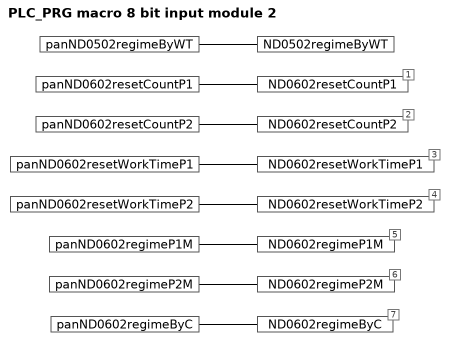
[picture p72: PLC_PRG macro 8 bit input module 2 (CFC)]
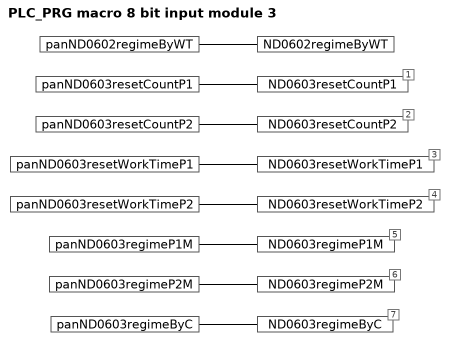
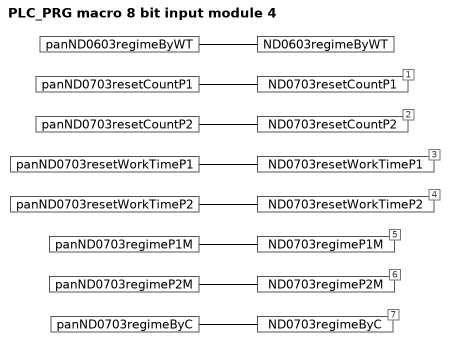
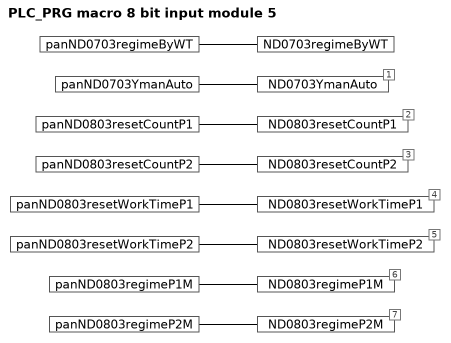
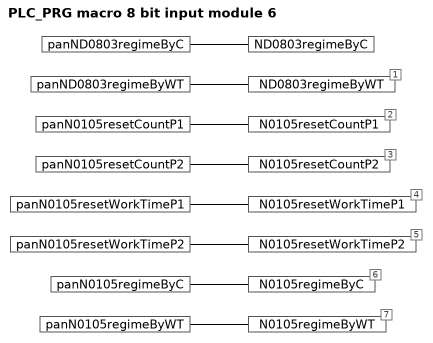
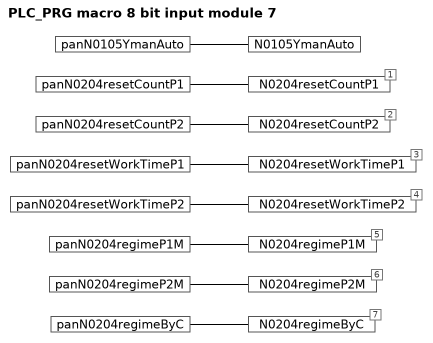
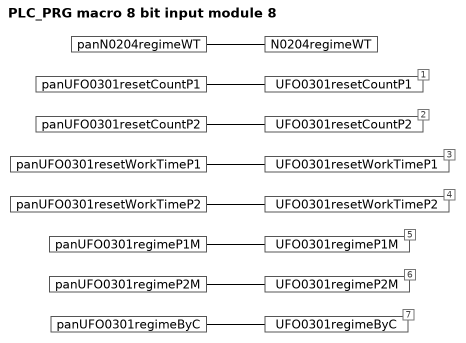
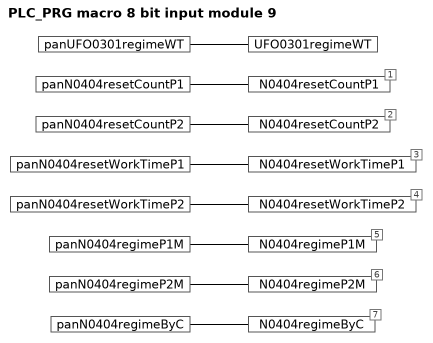
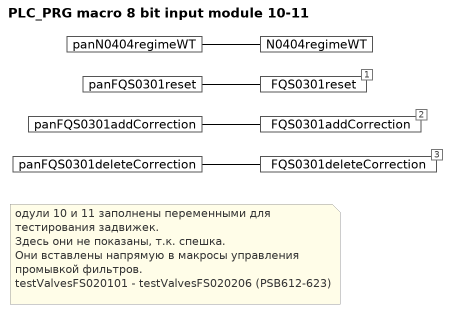
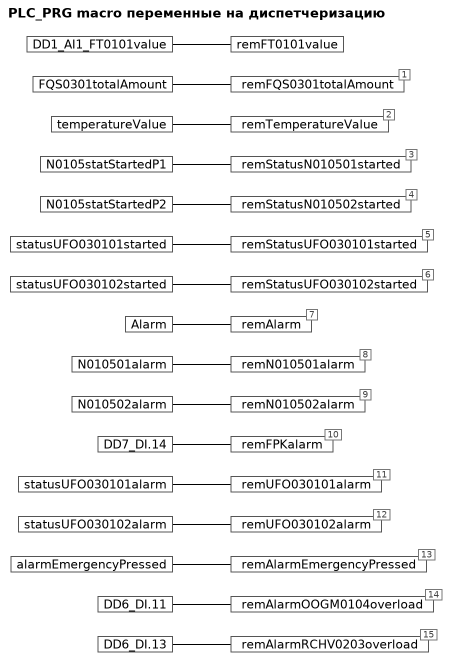
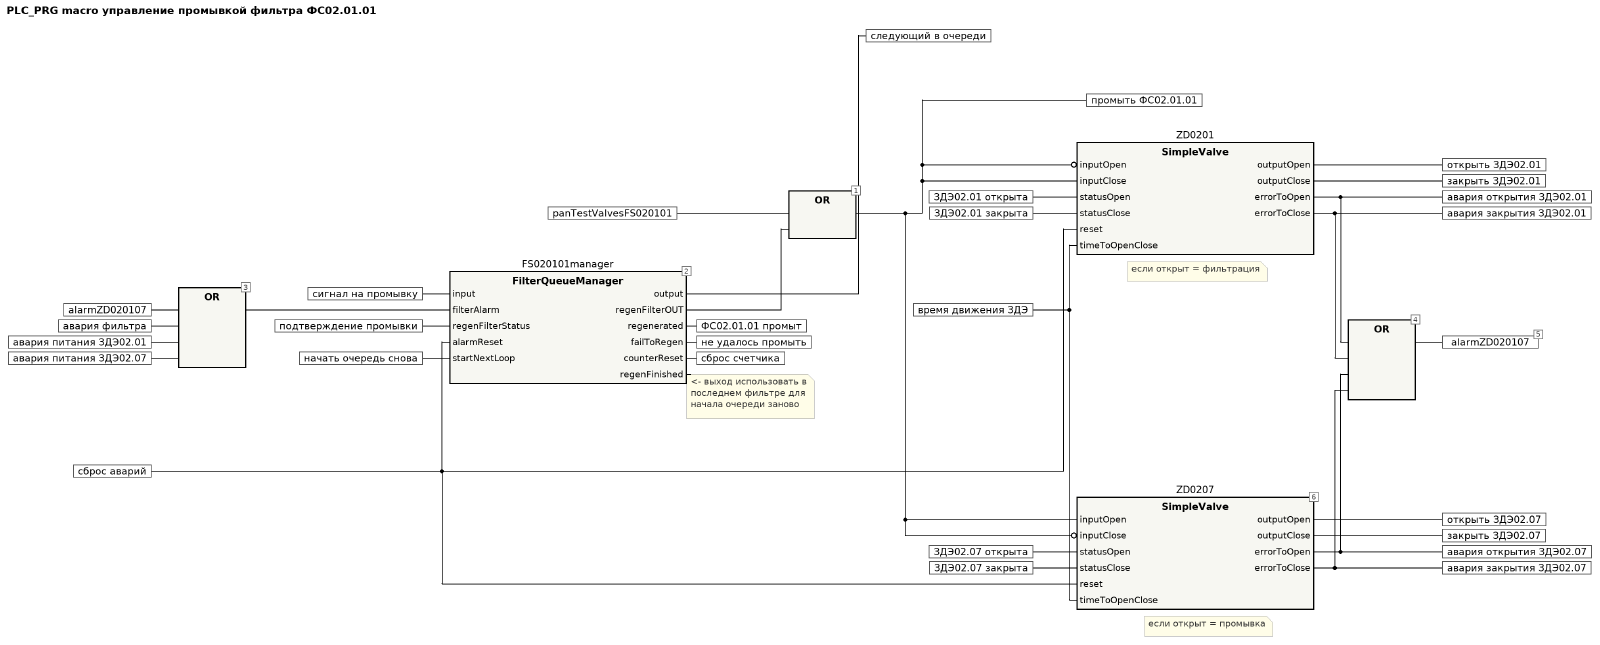
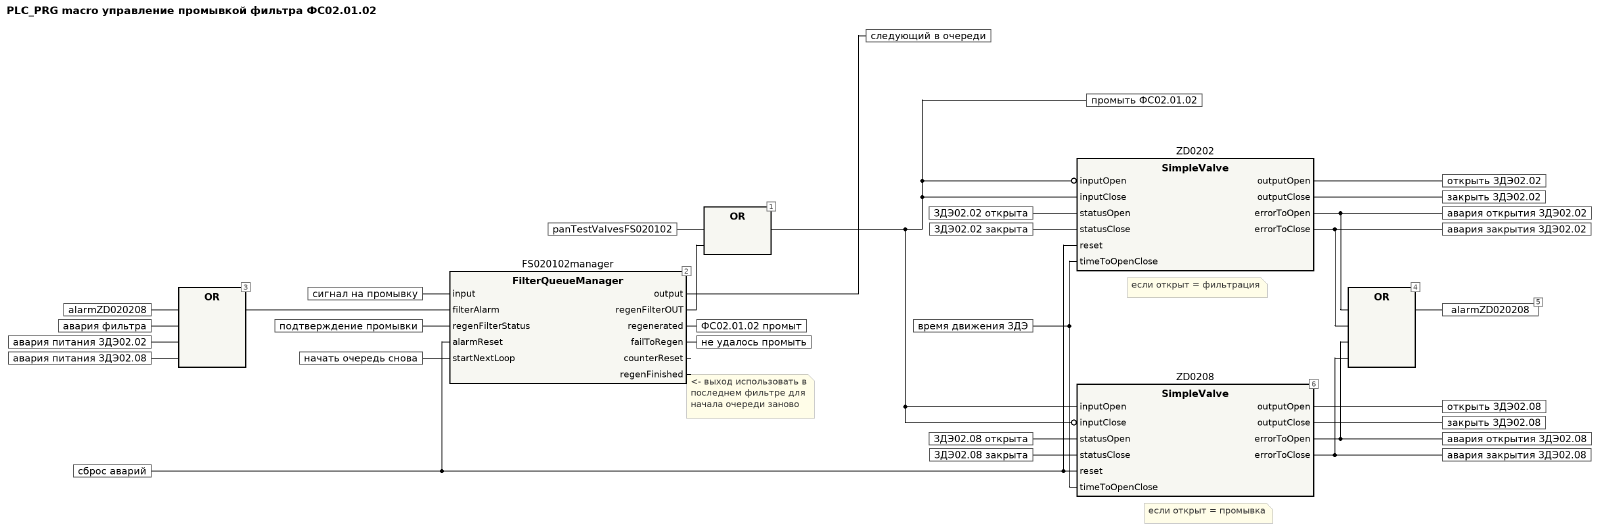
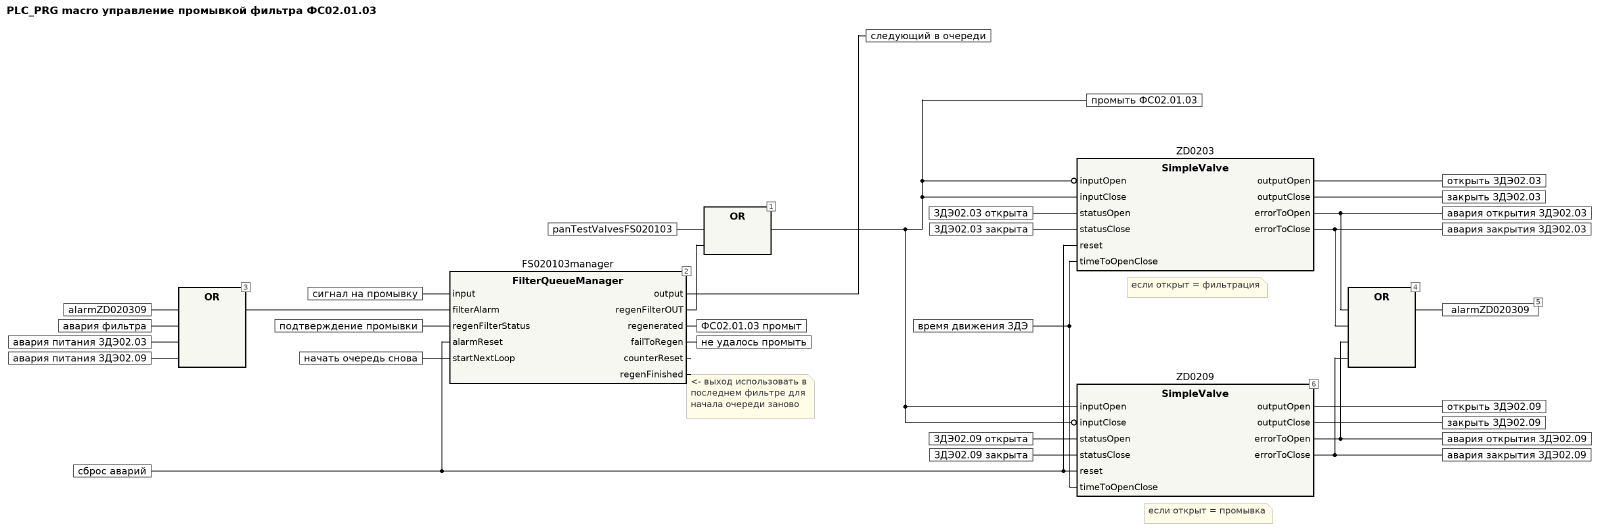
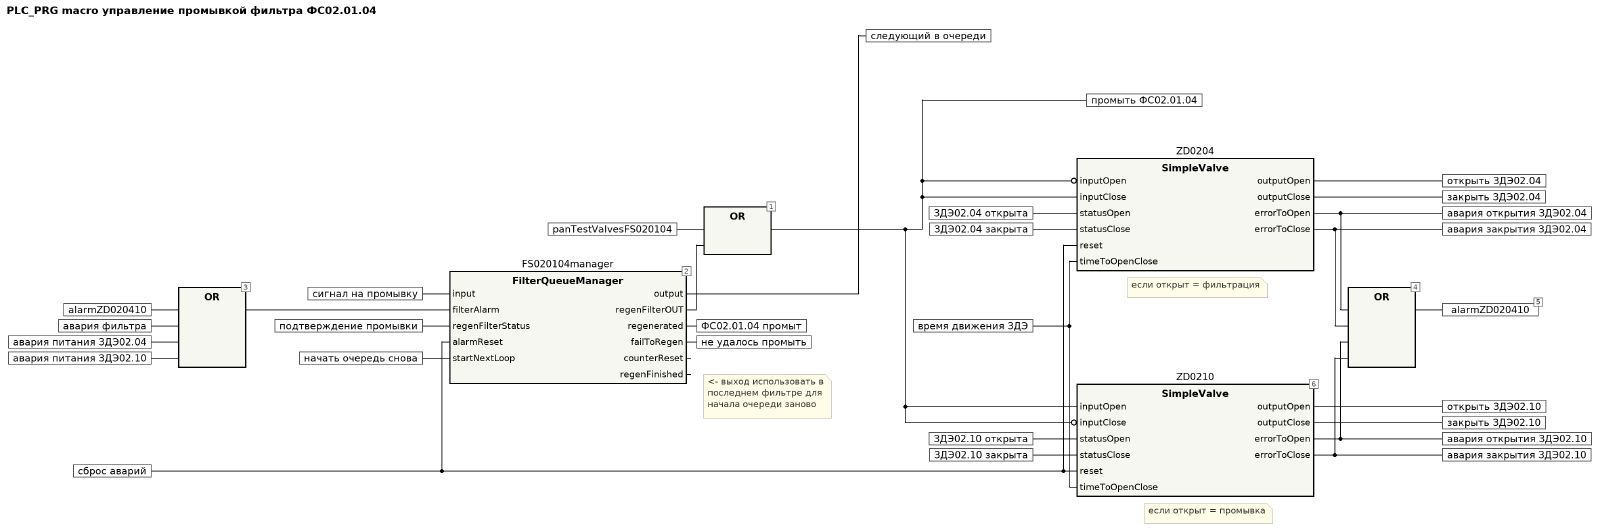
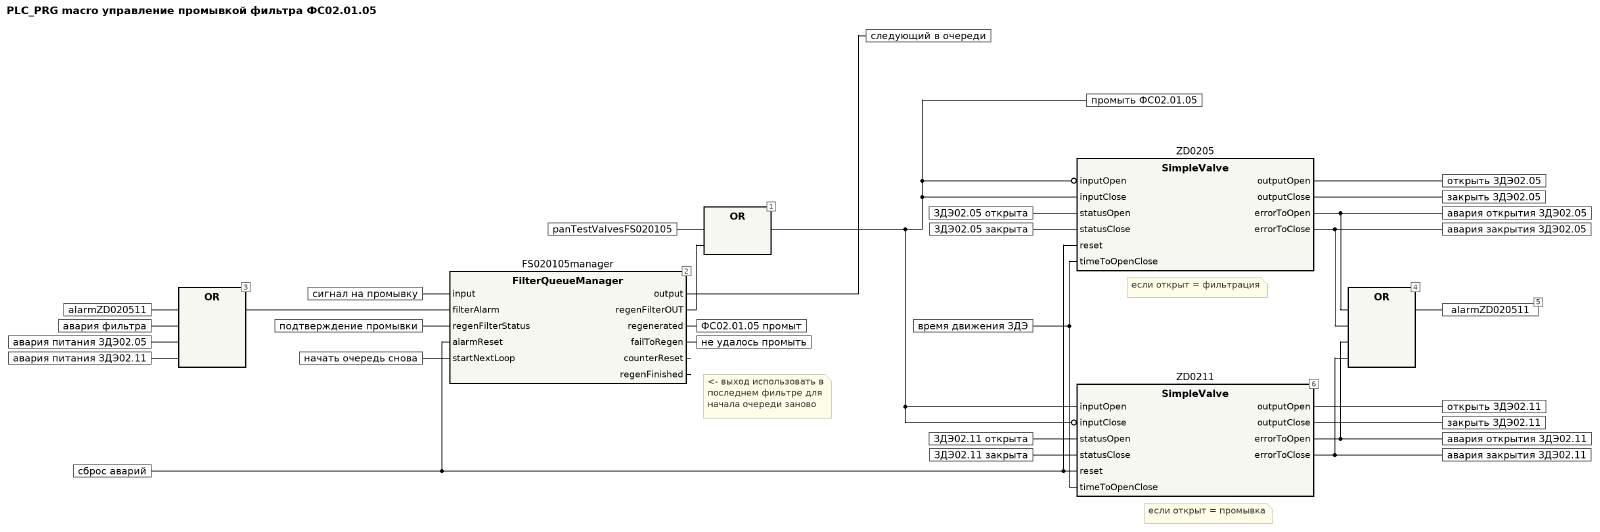
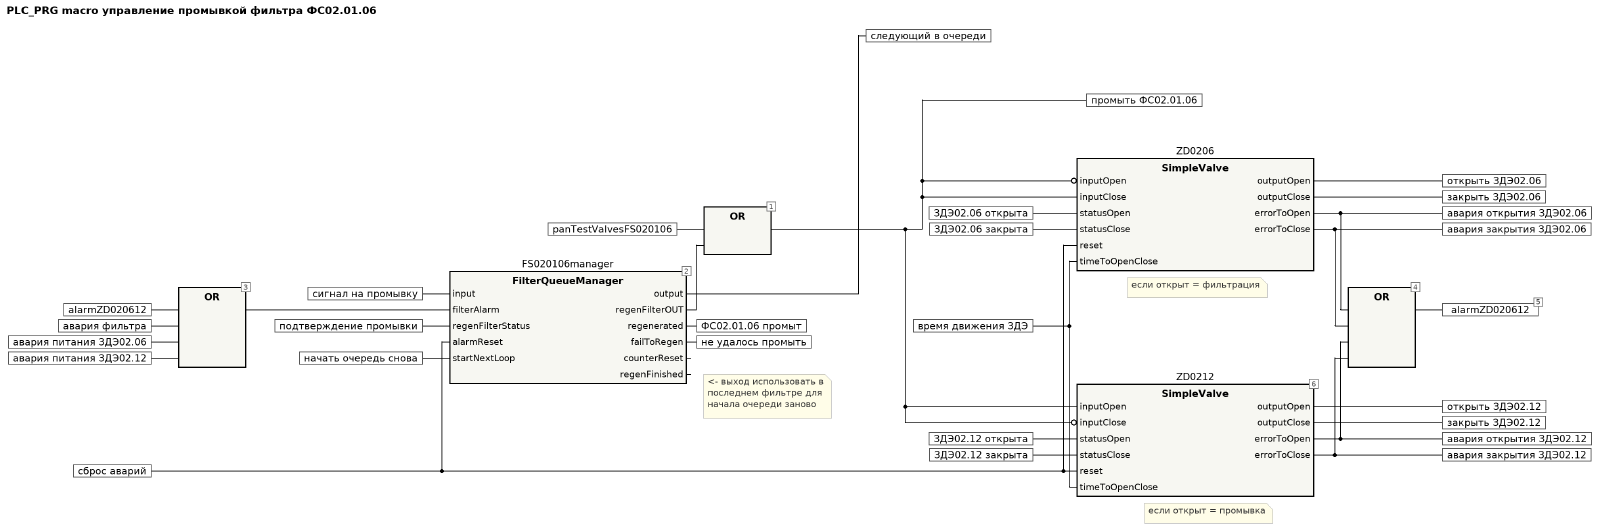
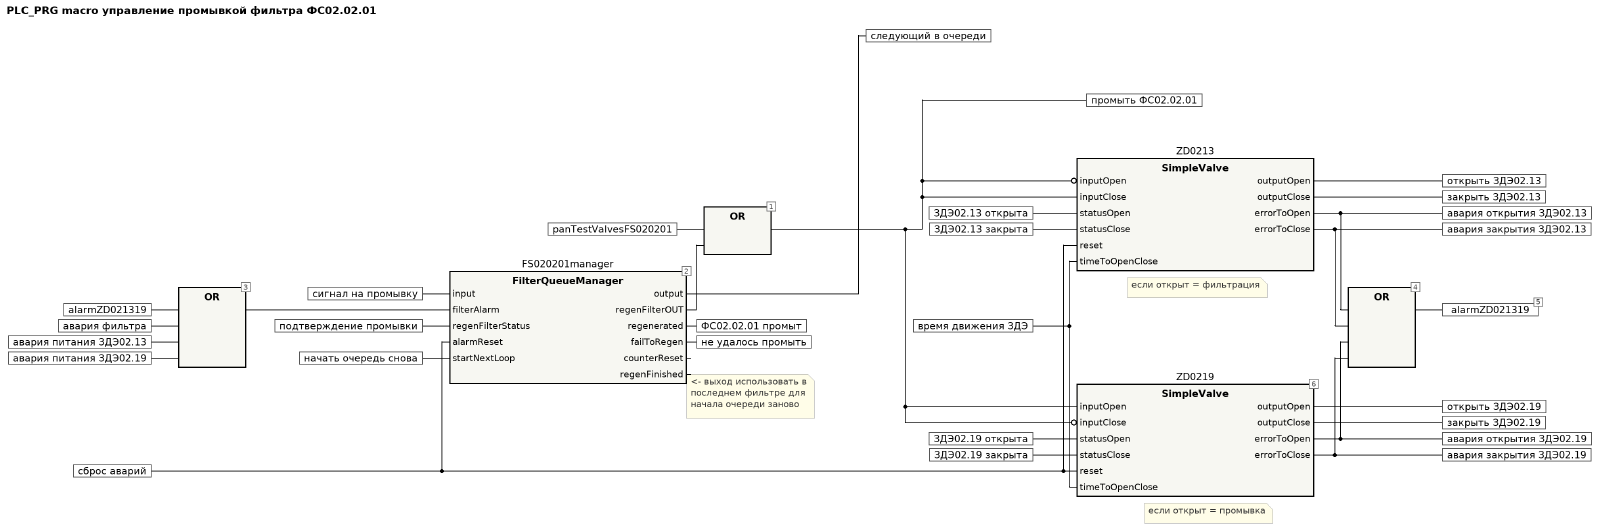
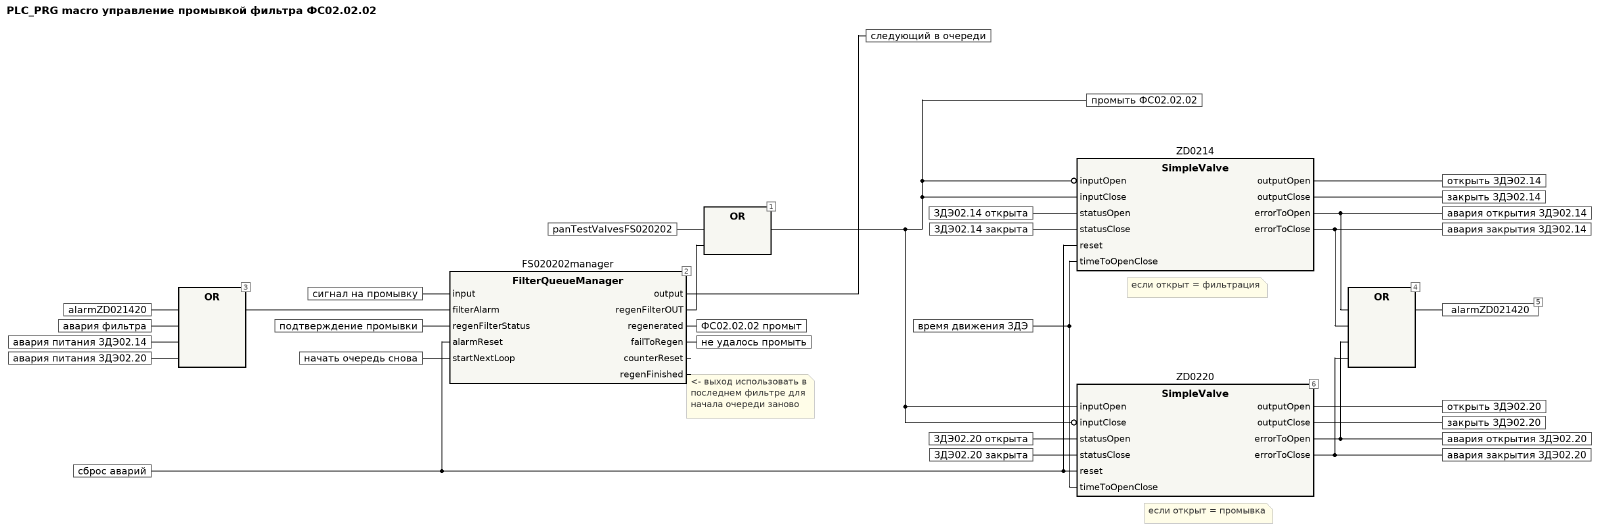
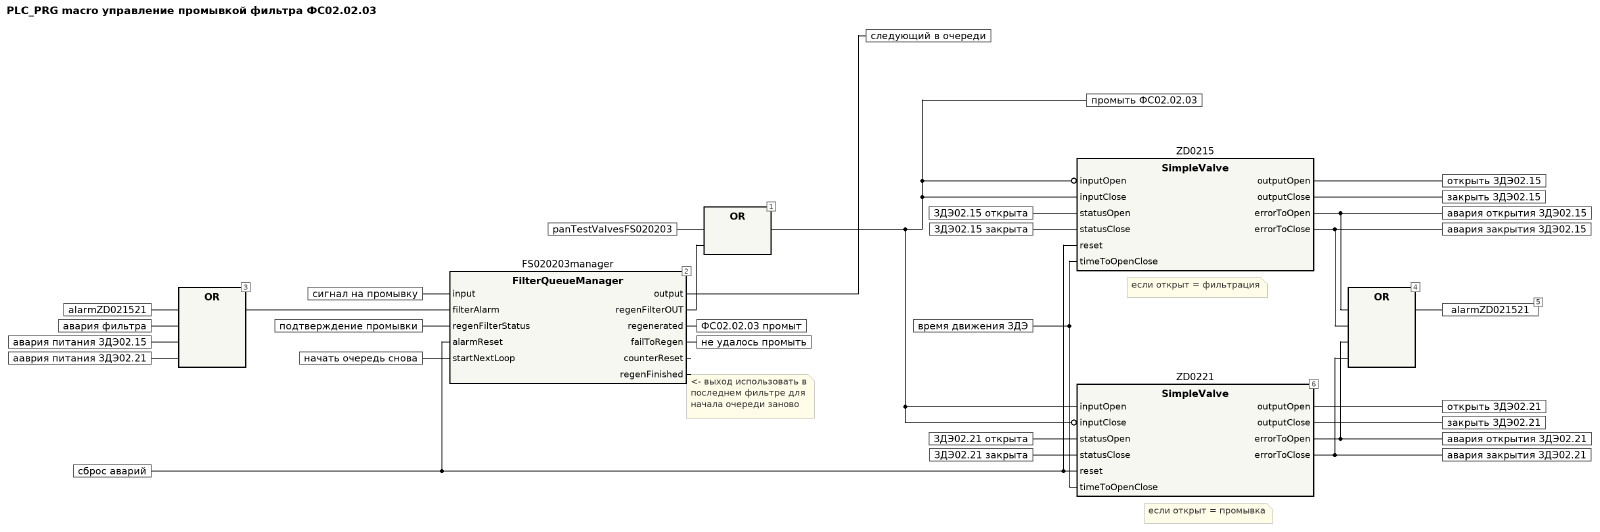
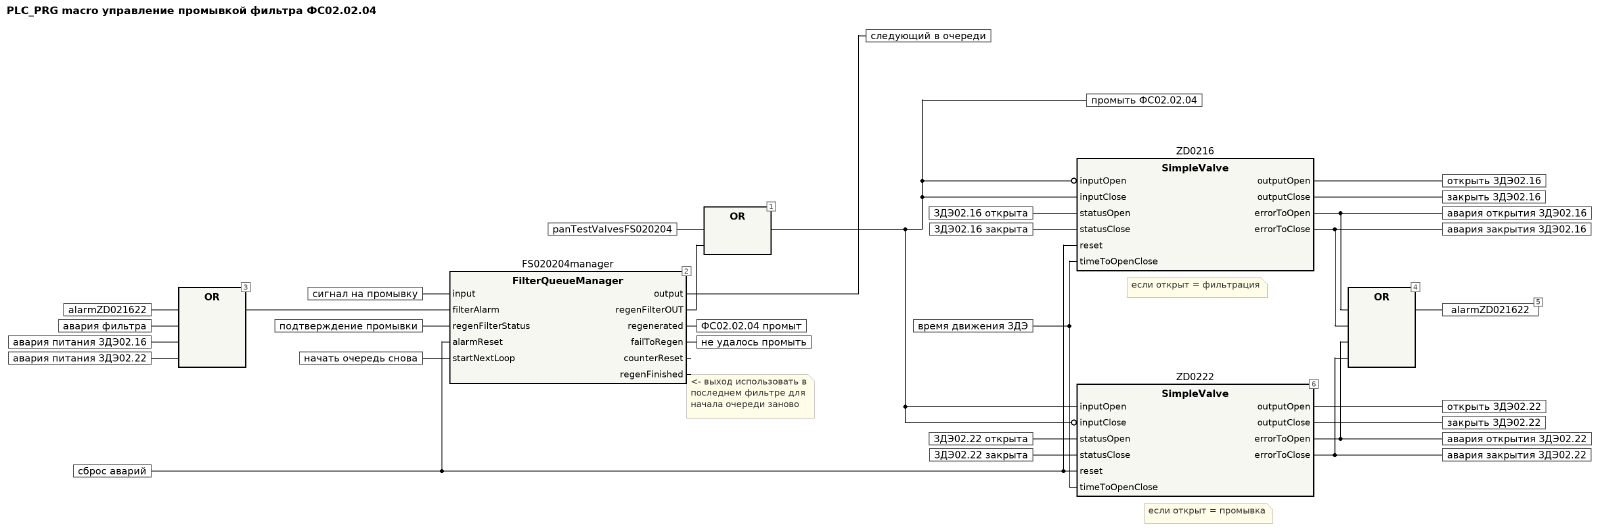
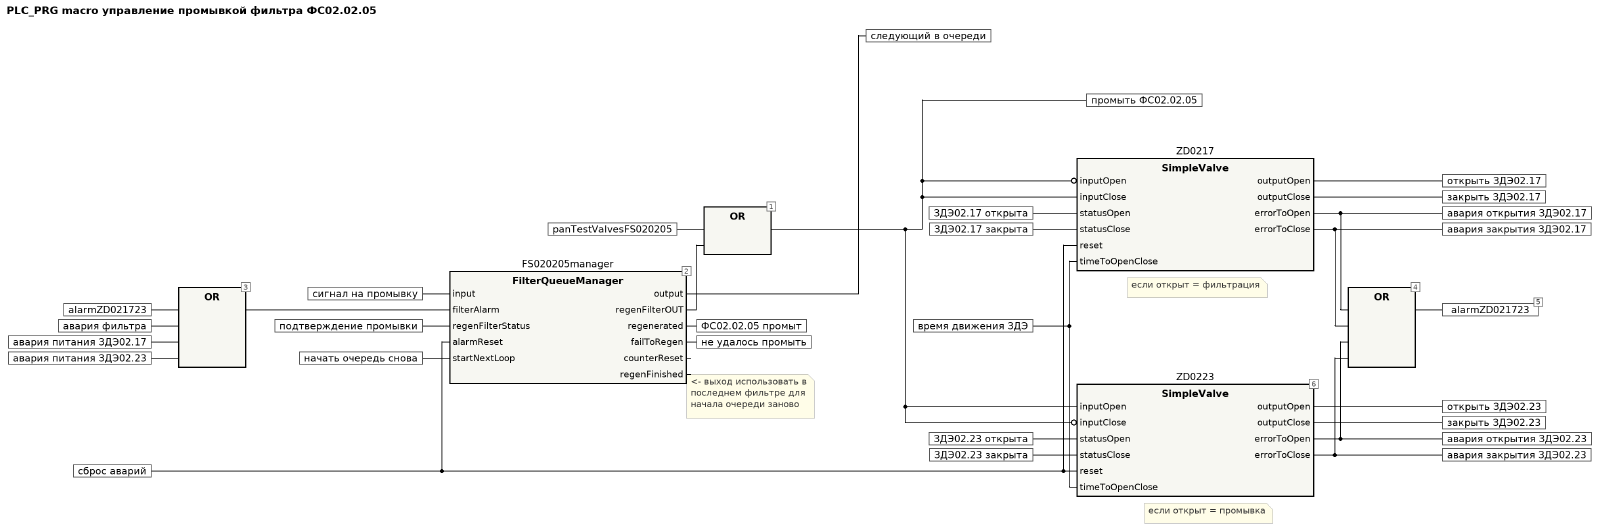
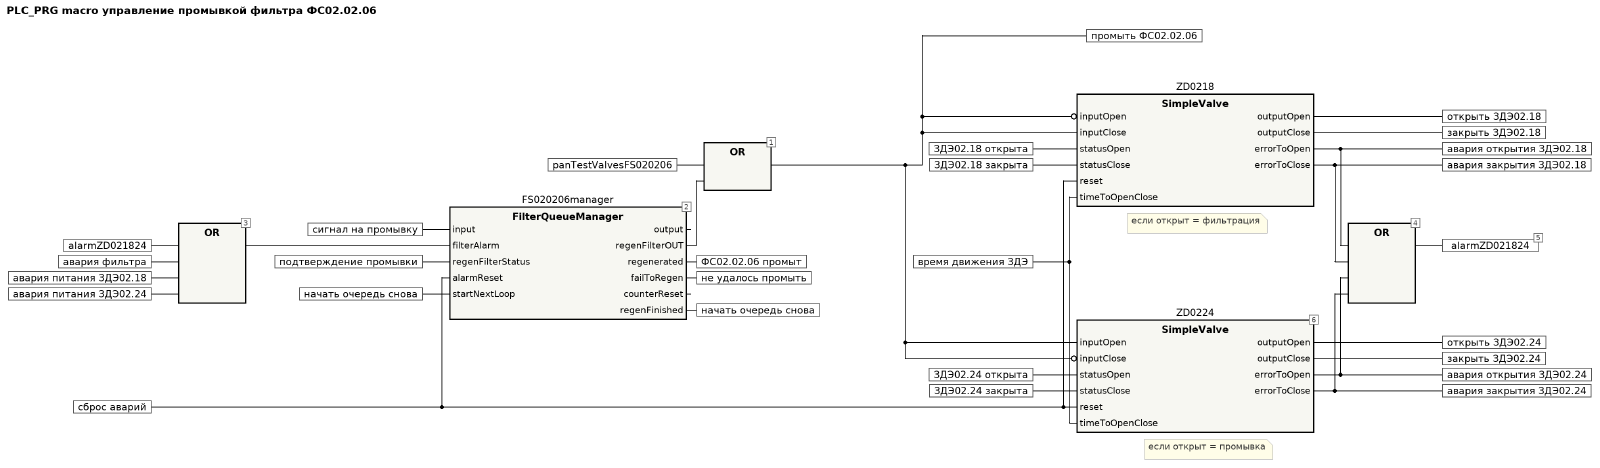
_CFC_ (* Continuous Function Chart, elements in execution order *)
(* 0 = перелив *)
(* авария обоих УФО, если проблемы / открытия/закрытия на одной из задвижек *)
(* авария питания ЗДЭ03.02 *)
(* авария питания ЗДЭ03.01 *)
(* статус-пуск Н01.05/02 *)
(* вкл КМ3 *)
(* Статус ПУСК / ЧРП Н01.05 *)
(* статус-пуск Н01.05/01 *)
(* вкл КМ2 *)
(* контроль обрыва или ошибок модулей в сети ПЛК *)
(* LSA01.02 перелив ОГМ01.04 *)
(* Нажат аварийный стоп. *)
(* авария сети (РКФ) *)
(* разрешение работы КНС / 1 = разрешено *)
(* Нажат аварийный стоп. *)
(* Блок управления разрешением работы КНС *)
(* авария сети (РКФ) *)
(* Авария питания клапанов КЭМ. *)
(* Авария питания розеток / управл.клапанов фильтров. *)
(* авария КНС *)
(* блок подачи сигнала на промывку *)
(* суммируем каждую секунду значение / мгновенного расхода в кубометрах в секунду *)
(* преобразуем расход из / кубометров в час в / кубометры в секунду *)
(* если есть расход / (больше нуля) *)
(* выдает импульс / каждую секунду *)
(* здесь мгновенный расход / в кубометрах в час (FT01.02) *)
(* Авария Н02.04/01 (0=авария) *)
(* Авария Н02.04/02 (0=авария) *)
(* промывка ФС02.01/06 *)
(* промывка ФС02.01/05 *)
(* промывка ФС02.01/04 *)
(* промывка ФС02.01/03 *)
(* промывка ФС02.01/02 *)
(* промывка ФС02.01/01 *)
(* пуск/стоп НД08.03/01 *)
(* пуск/стоп НД08.03/02 *)
(* пуск/стоп НД06.03/01 *)
(* пуск/стоп НД06.03/02 *)
(* пуск/стоп НД06.02/01 *)
(* пуск/стоп НД06.02/02 *)
(* пуск/стоп НД08.04 *)
(* пуск/стоп НД07.03/01 *)
(* пуск/стоп НД07.03/02 *)
(* авария М08.02 (УПФ) *)
(* авария М07.02 (УПЩ) *)
(* авария М06.04 (УПК) *)
(* работа М08.02 (УПФ) *)
(* работа М07.02 (УПЩ) *)
(* работа М06.04 (УПК) *)
(* Контроль, если УФО включили вручную, / а потока при этом нет. *)
(* авария УФО03.01/02 *)
(* работа УФО03.01/02 *)
(* авария УФО03.01/01 *)
(* Для подачи предостережения на пульте / оператора (при необходимости), а также / сигнализации лампой АВАРИЯ. *)
(* работа УФО03.01/01 *)
(* авария УФО03.01/02 *)
(* авария УФО03.01/01 *)
(* авария Н04.04/01 *)
(* авария Н04.04/02 *)
(* время контроля старта ФПК (по умолч.=3мин) *)
(* время работы ФПК после спада сигнала датч.осадка *)
(* запуск фильтрации *)
(* Защита от сухого хода насоса ФПК *)
(* датчик уровня осадка *)
(* Давление на входе ФПК (0...16 бар) *)
(* авария ФПК *)
(* подающий насос ФПК работает *)
(* ФПК готов к приему *)
(* ФПК не запустился *)
(* рН-метр QE01.02 на входе, / диапазон 0...14 *)
(* авария входа рН-метра QE01.01 *)
(* авария входа расходомера FT01.02 *)
(* расходомер FT01.01 на входе, / диапазон 0...600куб/час *)
(* авария НД08.04 *)
(* управление 4...20мА НД08.03/01 *)
(* пуск/стоп НД08.03/01 *)
(* пуск/стоп НД08.03/02 *)
(* управление 4...20мА НД08.03/02 *)
(* авария привода НД08.03/01 *)
(* авария привода НД08.03/02 *)
(* авария НД07.03/01 *)
(* авария НД07.03/02 *)
(* управление 4...20мА НД07.03/01 *)
(* управление 4...20мА НД07.03/02 *)
(* пуск/стоп НД07.03/01 *)
(* пуск/стоп НД07.03/02 *)
(* авария НД07.03/01 *)
(* авария НД07.03/02 *)
(* авария НД06.03/01 *)
(* авария НД06.03/02 *)
(* авария НД06.02/01 *)
(* авария НД06.02/02 *)
(* управление 4...20мА НД06.03/01 *)
(* пуск/стоп НД06.03/01 *)
(* пуск/стоп НД06.03/02 *)
(* управление 4...20мА НД06.03/02 *)
(* авария НД06.03/01 *)
(* авария НД06.03/02 *)
(* управление 4...20мА НД06.02/01 *)
(* пуск/стоп НД06.02/01 *)
(* пуск/стоп НД06.02/02 *)
(* управление 4...20мА НД06.02/02 *)
(* авария НД06.02/01 *)
(* авария НД06.02/02 *)
(* ошибка блока дозирования НД05.02 *)
(* авария входа датчика температуры *)
(* лампа АВАРИЯ *)
(* датчик температуры в помещении / (метран) диапазон: 0...+100С *)
(* управление 4...20мА НД05.02/01 *)
(* пуск/стоп НД05.02/01 *)
(* авария НД05.02/01 *)
(* авария НД05.02/02 *)
(* пуск/стоп НД05.02/02 *)
(* управление 4...20мА НД05.02/02 *)
(* АВАРИИ *)
(* авария привода НД08.03/01 *)
(* авария привода НД08.03/02 *)
(* авария НД08.04 *)
(* насос Н04.01 работает *)
(* пуск/стоп НД08.04 *)
(* управление 4...20мА НД08.04 *)
(* авария входа расходомера FT01.01 *)
(* расходомер FT01.02 на входе, / диапазон 0...600куб/час *)
(* рН-метр QE01.01 на входе, / диапазон 0...14 *)
(* авария входа рН-метра QE01.02 *)
(* сухой ход НД08.03/01 *)
(* сухой ход НД08.03/02 *)
(* сухой ход НД08.03/01 *)
(* сухой ход НД08.03/02 *)
(* LSA01.02 перелив ОГМ01.04 *)
(* Инициализирует требуемые булевые переменные / в момент старта выполнения программы. *)
(* Статус ПУСК ЧРП Н01.05 *)
(* LS01.03 - рабочий верхний уровень ОГМ01.04 автоматический пуск 01.05 *)
(* LS01.04 - нижний уровень ОГМ01.04, сухой ход Н01.05 *)
(* SA1 Ручной выбор Н01.05/01 = главный *)
(* SA1 Ручной выбор Н01.05/02 = главный *)
(* Стоп  Н01.05 (сброс самоподхвата реле) *)
(* время на создание потока *)
(* Пуск  Н01.05 *)
(* КМ1 питание ЧРП *)
(* КМ2 питание насоса 1 *)
(* КМ3 питание насоса 2 *)
(* Авария ЧРП Н01.05 *)
(* термоконтакт Н01.05/01 *)
(* термоконтакт Н01.05/02 *)
(* авария питания ЗДЭ02.25 *)
(* LSА02.01 Перелив РЧВ02.03 *)
(* Давление на входе ФПК / 0...16 бар (мах допуст.10) *)
(* Авария входа AI6 ПЛК, давл.ФПК *)
(* авария ФПК *)
(* Открыть КШЭ04.01 *)
(* статус КШЭ04.01 открыт *)
(* Закрыть КШЭ04.01 *)
(* статус КШЭ04.01 закрыт *)
(* подающий насос ФПК работает *)
(* стоп Н04.04 *)
(* пуск Н04.04/02 *)
(* пуск Н04.04/01 *)
(* авт.пуск Н04.04 *)
(* сухой ход Н04.04, 0=защита *)
(* авария Н04.04/01, 0=авария *)
(* авария Н04.04/02, 0=авария *)
(* импульсный расходомер *)
(* Авария Н02.04/01 (0=авария) *)
(* Авария Н02.04/02 (0=авария) *)
(* промывка ФС02.02/06 *)
(* промывка ФС02.02/05 *)
(* промывка ФС02.02/04 *)
(* промывка ФС02.02/03 *)
(* промывка ФС02.02/02 *)
(* промывка ФС02.02/01 *)
(* Клапан КЭМ05.01 открыт. *)
(* Клапан КЭМ06.01 открыт. *)
(* Клапан КЭМ07.01 открыт. *)
(* Клапан КЭМ08.01 открыт. *)
(* Сухой ход Н02.04 (LS02.03) 0=сух.ход *)
(* Стоп Н02.04 *)
(* Пуск Н02.04/01 *)
(* Пуск Н02.04/02 *)
(* текущий объем *)
(* заданный до промывки объем *)
(* 0=авария *)
(* авария (при 0) ФС02.01/06 *)
(* авария (при 0) ФС02.01/05 *)
(* авария (при 0) ФС02.01/04 *)
(* авария (при 0) ФС02.01/03 *)
(* авария (при 0) ФС02.01/02 *)
(* авария (при 0) ФС02.01/01 *)
(* авария (при 0) ФС02.02/06 *)
(* авария (при 0) ФС02.02/05 *)
(* авария (при 0) ФС02.02/04 *)
(* авария (при 0) ФС02.02/03 *)
(* авария (при 0) ФС02.02/02 *)
(* авария (при 0) ФС02.02/01 *)
(* сброс счетчика стоков до следующей промывки *)
(* подсчет общего объема стоков, прошедшего через расходомер FT01.02 *)
(* очередь передается на 2 ступень *)
(* авария питания ЗДЭ02.01 *)
(* авария питания ЗДЭ02.02 *)
(* авария питания ЗДЭ02.03 *)
(* авария питания ЗДЭ02.04 *)
(* авария питания ЗДЭ02.05 *)
(* авария питания ЗДЭ02.06 *)
(* авария питания ЗДЭ02.07 *)
(* авария питания ЗДЭ02.08 *)
(* авария питания ЗДЭ02.09 *)
(* авария питания ЗДЭ02.10 *)
(* авария питания ЗДЭ02.11 *)
(* авария питания ЗДЭ02.12 *)
(* авария питания ЗДЭ02.13 *)
(* авария питания ЗДЭ02.14 *)
(* авария питания ЗДЭ02.15 *)
(* авария питания ЗДЭ02.16 *)
(* авария питания ЗДЭ02.17 *)
(* авария питания ЗДЭ02.18 *)
(* авария питания ЗДЭ02.19 *)
(* авария питания ЗДЭ02.20 *)
(* авария питания ЗДЭ02.21 *)
(* авария питания ЗДЭ02.22 *)
(* авария питания ЗДЭ02.23 *)
(* авария питания ЗДЭ02.24 *)
(* инвертирование сигнала, чтобы все аварии / обозначались как 1 (TRUE) *)
(* авария НД05.02/01 *)
(* авария НД05.02/02 *)
(* авария питания КШЭ04.01 *)
(* 1=открыть; 0 = закрыть *)
(* в этом макросе лежит управление режимом тестирования задвижек ЗДЭ03 / Тестирование запрещает автоматический запуск УФО от ПЛК *)
#0 rTrigStartInitializer:R_TRIG(CLK: TRUE)
#1 startInitializer <= #0.Q
#2 MACRO контроль температуры в помещении(pin 1 "вход датчика температуры": DD1_AI0, pin 2 "минимально допустимая температура в помещении": maxTemperature, pin 3 "максимально допустимая температура в помещении": minTemperature)
	(* задаем границы допустимой температуры в помещении / проверяем что измеренное значение в заданном диапазоне *)
	(* не смотрим конкретный тип ошибки / (работает не точно, обрыв определяет как слишком маленькое значение) / если не равно 0 - значит на входе ошибка *)
	#3 DD1_AI0_temperature:DECODE_FLOAT(VALUE: pin 1, DEF_VALUE: -)
	#4 NE(#3._ERR, 0)
	out 2 "авария датчика температуры" <= #4
	out 1 "температура в помещении" <= #3.OUT_VALUE
	#5 REAL_TO_INT(#3.OUT_VALUE)
	#6 temperatureLimits:LIMITALARM(IN: #5, HIGH: pin 3, LOW: pin 2)
	out 3 "температура выше заданного диапазона" <= #6.O
	out 4 "температура ниже заданного диапазона" <= #6.U
	#7 temperatureLimits:LIMITALARM(IN: -, HIGH: -, LOW: -)
END_MACRO
#8 temperatureValue <= #2.out 1
#9 DD1_AI0_error <= #2.out 2
#10 alarmHighTemperature <= #2.out 3
#11 alarmLowTemperature <= #2.out 4
#12 OR(testKSHE0401, DD7_DI.13)
#13 MACRO клапан шаровый перед ФПК (КШЭ04.01)(pin 1 "сигнал "подающий насос ФПК" работает": #12, pin 2 "статус КШЭ04.01 открыт": DD9_DI.2, pin 3 "статус КШЭ04.01 закрыт": DD9_DI.3, pin 4 "сброс аварий": alarmReset, pin 5 "время на открытие/закрытие": timeToOpenCloseValve)
	#14 FPKkshe0401DelayToOpen:TON(IN: #16.outputOpen, PT: T#1s)
	out 1 "выход на открытие КШЭ04.01" <= #14.Q
	#15 FPKkshe0401DelayToClose:TON(IN: #16.outputClose, PT: T#1s)
	out 2 "выход на закрытие КШЭ04.01" <= #15.Q
	#16 FPKkshe0401:SimpleValve(inputOpen: pin 1, inputClose: #17, statusOpen: pin 2, statusClose: pin 3, reset: pin 4, timeToOpenClose: pin 5)
	#17 NOT(pin 1)
	out 3 "авария на открытие КШЭ04.01" <= #16.errorToOpen
	out 4 "авария на закрытие КШЭ04.01" <= #16.errorToClose
END_MACRO
#18 DD4_DO.2 <= #13.out 1
#19 DD4_DO.3 <= #13.out 2
#20 FPKkshe0401errorToOpen <= #13.out 3
#21 FPKkshe0401errorToClose <= #13.out 4
#22 OR(DD1_AI0_error, DD1_AI1_error, DD1_AI2_error, DD1_AI3_error, DD1_AI4_error, alarmHighTemperature, alarmLowTemperature, ND0502dosingError, ND0602dosingError, ND0603dosingError, ND0803dosingError, ND0804dosingError, DD1_DI6, DD1_DI7, N010501alarm, N010502alarm, ZDE0225errorToOpen, ZDE0225errorToClose, DD7_DI.14, FPKnotStarted, DD1_AI5_error, FPKkshe0401errorToOpen, FPKkshe0401errorToClose, DD5_DI.27, DD5_DI.29, filterFailToRegen020101, errorToOpenZD0201, errorToCloseZD0201, errorToOpenZD0207, errorToCloseZD0207, filterFailToRegen020102, errorToOpenZD0202, errorToCloseZD0202, errorToOpenZD0208, errorToCloseZD0208, filterFailToRegen020103, errorToOpenZD0203, errorToCloseZD0203, errorToOpenZD0209, errorToCloseZD0209, filterFailToRegen020104, errorToOpenZD0204, errorToCloseZD0204, errorToOpenZD0210, errorToCloseZD0210, filterFailToRegen020105, errorToOpenZD0205, errorToCloseZD0205, errorToOpenZD0211, errorToCloseZD0211, filterFailToRegen020106, errorToOpenZD0206, errorToCloseZD0206, errorToOpenZD0212, errorToCloseZD0212, filterFailToRegen020201, errorToOpenZD0213, errorToCloseZD0213, errorToOpenZD0219, errorToCloseZD0219, filterFailToRegen020202, errorToOpenZD0214, errorToCloseZD0214, errorToOpenZD0220, errorToCloseZD0220, filterFailToRegen020203, errorToOpenZD0215, errorToCloseZD0215, errorToOpenZD0221, errorToCloseZD0221, filterFailToRegen020204, errorToOpenZD0216, errorToCloseZD0216, errorToOpenZD0222, errorToCloseZD0222, filterFailToRegen020205, errorToOpenZD0217, errorToCloseZD0217, errorToOpenZD0223, errorToCloseZD0223, filterFailToRegen020206, errorToOpenZD0218, errorToCloseZD0218, errorToOpenZD0224, errorToCloseZD0224, alarmPLKnetwork, alarmND050201, alarmND050202, alarmND060201, alarmND060202, alarmND060301, alarmND060302, alarmND070301, alarmND070302, alarmND080301, alarmND080302, alarmND0804, alarmOGM0104overload, alarmRCHV0203overload, alarmN040402, alarmN040401, alarmM0604, alarmM0702, alarmM0802, alarmN020401, alarmN020402, alarmFS020101, alarmFS020102, alarmFS020103, alarmFS020104, alarmFS020105, alarmFS020106, alarmFS020201, alarmFS020202, alarmFS020203, alarmFS020204, alarmFS020205, alarmFS020206, alarmZDE0201power, alarmZDE0202power, alarmZDE0203power, alarmZDE0204power, alarmZDE0205power, alarmZDE0206power, alarmZDE0207power, alarmZDE0208power, alarmZDE0209power, alarmZDE0210power, alarmZDE0211power, alarmZDE0212power, alarmZDE0213power, alarmZDE0214power, alarmZDE0215power, alarmZDE0216power, alarmZDE0217power, alarmZDE0218power, alarmZDE0219power, alarmZDE0220power, alarmZDE0221power, alarmZDE0222power, alarmZDE0223power, alarmZDE0224power, alarmZDE0225power, alarmKSHE0401power, alarmKNS, alarmPowerSocketFS, alarmKEMvalvesPower, alarmEmergencyPressed, alarmRKF, errorToOpenZDE0301, errorToCloseZDE0301, errorToOpenZDE0302, errorToCloseZDE0302, alarmZDE0301power, alarmZDE0302power)
#23 DD1_DO11 <= #22
#24 alarm <= #22
#25 MACRO контроль аналогового входа DD1_AI1(pin 1 "вход": DD1_AI1)
	(* Не смотрим конкретную ошибку, / определяем,что вход неисправен без расшифровки. *)
	#26 DD1_AI1_FT0101:DECODE_FLOAT(VALUE: pin 1, DEF_VALUE: -)
	#27 NE(#26._ERR, 0)
	out 2 "авария" <= #27
	out 1 "выход" <= #26.OUT_VALUE
END_MACRO
#28 DD1_AI1_FT0101value <= #25.out 1
#29 DD1_AI1_error <= #25.out 2
#30 MACRO контроль аналогового входа DD1_AI2(pin 1 "вход": DD1_AI2)
	(* Не смотрим конкретную ошибку, / определяем,что вход неисправен без расшифровки. *)
	#31 DD1_AI2_FT0102:DECODE_FLOAT(VALUE: pin 1, DEF_VALUE: -)
	#32 NE(#31._ERR, 0)
	out 2 "авария" <= #32
	out 1 "выход" <= #31.OUT_VALUE
END_MACRO
#33 DD1_AI2_FT0102value <= #30.out 1
#34 DD1_AI2_error <= #30.out 2
#35 MACRO управление Н01.05 (поддержание заданного расхода по FT01.02)(pin 1 "статус ПУСК ЧРП (реле)": DD5_DI.4, pin 2 "LS01.03 раб.уров.": DD6_DI.12, pin 3 "LS01.04 ниж.уров.(сух.ход)": DD5_DI.0, pin 4 "SA1ручной выб.Н01.05/01-главный": DD5_DI.5, pin 5 "SA1ручной выб.Н01.05/02-главный": DD5_DI.6, pin 6 "включить режим "по кол.вкл."": N0105regimeByC, pin 7 "включить режим "по наработке"": N0105regimeByWT, pin 8 "значение расхода от FT01.02": DD1_AI2_FT0102value, pin 9 "уставка расхода": N0105flowSetValue, pin 10 "время на создание потока": N0105minFlowTime, pin 11 "Р-коэфф.": N0105koeffP, pin 12 "I-коэфф": N0105koeffI, pin 13 "Д-коэфф": N0105koeffD, pin 14 "управление ЧРП в ручн.реж.(4...20мА)": N0105YoutManual, pin 15 "переключатель управление ЧРП РУЧН/АВТ": N0105YmanAuto, pin 16 "мин.допустимый расход": N0105minFlow, pin 17 "термоконтакт Н01.05/01": DD5_DI.2, pin 18 "термоконтакт Н01.05/02": DD5_DI.3, pin 19 "авария ЧРП Н01.05": DD5_DI.1, pin 20 "сброс аварии": alarmReset, pin 21 "сброс кол-ва вкл.Н01.05/01": N0105resetCountP1, pin 22 "сброс кол-ва вкл.Н01.05/02": N0105resetCountP2, pin 23 "сброс наработки Н01.05/01": N0105resetWorkTimeP1, pin 24 "сброс наработки Н01.05/02": N0105resetWorkTimeP2)
	(* время на создание потока *)
	(* Пуск  Н01.05 *)
	(* режимы по количеству включений,  или по наработке / активны если оба входа SA1 не активны *)
	(* управление Н01.05 - поддержание / заданного расхода по FT01.02 *)
	(* по умолчанию при старте программы *)
	(* если на входе true / то нижнее значение, / иначе то, что посередине *)
	(* Если насос создает давление меньше / указанного, то авария. *)
	#36 OR(pin 2, #37.Q)
	#37 N0105startTrig:R_TRIG(CLK: pin 1)
	#38 N0105stopTrig:F_TRIG(CLK: pin 1)
	#39 N0105startTrigg:RS(SET: #36, RESET1: #41)
	#40 N0105regime:choosePumpRegime(start: #39.Q1, pump1Main: pin 4, pump2Main: pin 5, byCounter: #44, byWorkTime: #50)
	out 2 "статус режим "Н01.05/01 - главный"" <= #40.pump1MainActive
	out 3 "статус режим "Н01.05/02 - главный"" <= #40.pump2MainActive
	out 4 "статус режим "по кол-ву вкл."" <= #40.byCounterActive
	#41 OR(#38.Q, #42)
	out 5 "статус режим "по наработке"." <= #40.byWorkTimeActive
	#42 NOT(pin 3)
	#43 NOT(#39.Q1)
	out 1 "СТОП (сброс самоподхвата реле пуска ЧРП)." <= #43
	#44 AND(NOT pin 4, NOT pin 5, #47.Q1)
	#45 OR(pin 6, startInitializer)
	#46 N0105regByCinit:R_TRIG(CLK: #45)
	#47 N0105regByCtrig:RS(SET: #46.Q, RESET1: #55.Q)
	#48 N0105twoPumpOneDriveManager:TwoPumpOneDriveManager(startStopPump1: #40.startPump1, startStopPump2: #40.startPump2, alarmPump1: N010501alarm, alarmPump2: N010502alarm, alarmReset: alarmReset, counterStart: #40.startByCounter, Pump1ResetCounter: pin 21, Pump2ResetCounter: pin 22, ValueToResetCounter: -, workTimeStart: #40.startByWorkTime, workTimePump1Reset: pin 23, workTimePump2Reset: pin 24, timeKM1off: -, timeKM23DelayON: -, timeKM23offDelay: -, timeReadyToStartDelay: -)
	out 6 "кол-во включений Н01.05/01" <= #48.counterPump1
	#49 AND(#48.pump1active, #65)
	out 7 "кол-во включений Н01.05/02" <= #48.counterPump2
	out 8 "наработка Н01.05/01" <= #48.currentWorkTimePump1
	out 15 "авария Н01.05/01" <= #53.Q1
	#50 AND(NOT pin 4, NOT pin 5, #56.Q1)
	out 9 "наработка Н01.05/02" <= #48.currentWorkTimePump2
	out 10 "КМ1-питание ЧРП" <= #48.DriveKM
	#51 AND(#48.pump1active, #57)
	#52 OR(#49, #51)
	#53 N010501alarmTrig:RS(SET: #52, RESET1: pin 20)
	#54 N010501alarm <= #53.Q1
	#55 N0105regWTinit:R_TRIG(CLK: pin 7)
	#56 N0105regWTtrig:RS(SET: #55.Q, RESET1: #46.Q)
	out 11 "КМ2-питание Н01.05/01" <= #48.pump1KM
	out 12 "КМ3-питание Н01.05/02" <= #48.pump2KM
	#57 OR(NOT pin 17, NOT pin 19)
	out 13 "пуск ЧРП (Н01.05)" <= #48.driveStart
	#58 OR(NOT pin 19, NOT pin 18)
	out 16 "авария Н01.05/02" <= #61.Q1
	#59 AND(#58, #48.pump2active)
	#60 OR(#59, #63)
	#61 N010502alarmTrig:RS(SET: #60, RESET1: pin 20)
	#62 N010502alarm <= #61.Q1
	#63 AND(#48.pump2active, #65)
	#64 N0105timerminFlow:TON(IN: #48.driveStart, PT: pin 10)
	#65 AND(#64.Q, #66)
	#66 LE(pin 8, pin 16)
	#67 SEL(#48.driveStart, 0, #68.Y)
	out 14 "управление ЧРП (4...20мА)" <= #67
	#68 N0105pidReg:PID(ACTUAL: pin 8, SET_POINT: pin 9, KP: pin 11, TN: pin 12, TV: pin 13, Y_MANUAL: pin 14, Y_OFFSET: -, Y_MIN: 4, Y_MAX: 20, MANUAL: pin 15, RESET: #68.OVERFLOW)
END_MACRO
#69 DD4_DO.13 <= #35.out 1
#70 N0105statRegimeP1M <= #35.out 2
#71 N0105statRegimeP2M <= #35.out 3
#72 N0105statRegimeByC <= #35.out 4
#73 N0105statRegimeByWT <= #35.out 5
#74 N0105counterP1 <= #35.out 6
#75 N0105counterP2 <= #35.out 7
#76 N0105workTimeP1 <= #35.out 8
#77 N0105workTimeP2 <= #35.out 9
#78 DD2_DO.0 <= #35.out 10
#79 DD2_DO.1 <= #35.out 11
#80 DD2_DO.2 <= #35.out 12
#81 DD1_DO0 <= #35.out 13
#82 DD1_AO0 <= #35.out 14
#83 N010501alarm <= #35.out 15
#84 N010502alarm <= #35.out 16
#85 MACRO Сигналы работы с ФП04.02 (фильтр-пресс)(pin 1 "датчик уровня осадка": DD7_DI.15, pin 2 "время работы ФПК (после выкл.датч.осадка)": FPKtimeToWork, pin 3 "защита от сухого хода": DD6_DI.10, pin 4 "ошибка входа AI (обрыв)": DD1_AI5_error, pin 5 "авария ФПК": DD7_DI.14, pin 6 "фильтр-пресс готов к приему": DD7_DI.12, pin 7 "давление на входе в ФПК": DD1_AI5_FPKpressureValue, pin 8 "мах допустимое давление": FPKmaxPressureValue, pin 9 "подающий насос ФПК работает": DD7_DI.13, pin 10 "время контроля старта ФПК": FPKnotStartedTime, pin 11 "сброс аварий": alarmReset)
	(* ФПК готов к приему осадка *)
	(* LS01.01-нижн.уровень на входе ОГМ01.04 / защита от сух. хода насоса ФПК *)
	(* LES01.01-сигнал датчика уровня осадка ОГМ01.04 / запуск процесса фильтрации *)
	(* Время работы ФПК после / спада сигнала уровня осадка / по умолч.15мин. *)
	(* Давление на входе ФПК / 0...16 бар (мах допуст.10) *)
	(* максимально допустимое давление / на входе ФПК *)
	(* Условие сброса сигнала о грязном фильтр-прессе: / 1. Пропал сигнал о готовности ФПК; / 2. Появился сигнал о готовности ФПК. / Это значит, что оператор раздвигал плиты, / чистил и снова сдвигал их. *)
	#86 FPKneedToCleanResetFtrig:F_TRIG(CLK: FPKneedToCleanReset)
	#87 FPKstartTrig:RS(SET: pin 1, RESET1: #93)
	out 1 "запуск/старт ФПК" <= #87.Q1
	#88 FPKstopTimer:TOF(IN: pin 1, PT: pin 2)
	#89 FPKstopFtrig:F_TRIG(CLK: #88.Q)
	#90 AND(#87.Q1, #91)
	#91 NOT(pin 11)
	#92 AND(#87.Q1, #94.Q, #96)
	out 2 "ФПК не стартовал" <= #92
	#93 OR(#89.Q, pin 4, pin 5, #95, #97, #100.Q1)
	#94 FPKnotStartedTimer:TON(IN: #90, PT: pin 10)
	#95 NOT(pin 3)
	#96 NOT(pin 9)
	#97 NOT(pin 6)
	#98 AND(#87.Q1, #99)
	#99 GE(pin 7, pin 8)
	#100 FPKneedToCleanTrig:RS(SET: #98, RESET1: #86.Q)
	out 3 "ФПК нужно почистить!" <= #100.Q1
	#101 S FPKneedToCleanReset <= #100.Q1
	#102 FPKneedToCleanResetRtrig:R_TRIG(CLK: pin 6)
	#103 R FPKneedToCleanReset <= #102.Q
END_MACRO
#104 DD1_DO10 <= #85.out 1
#105 FPKnotStarted <= #85.out 2
#106 FPKneedToClean <= #85.out 3
#107 MACRO контроль аналогового входа DD1_AI3(pin 1 "вход": DD1_AI3)
	(* Не смотрим конкретную ошибку, / определяем,что вход неисправен без расшифровки. *)
	#108 DD1_AI3_QE0101:DECODE_FLOAT(VALUE: pin 1, DEF_VALUE: -)
	#109 NE(#108._ERR, 0)
	out 2 "авария" <= #109
	out 1 "выход" <= #108.OUT_VALUE
END_MACRO
#110 DD1_AI3_QE0101value <= #107.out 1
#111 DD1_AI3_error <= #107.out 2
#112 MACRO контроль аналогового входа DD1_AI4(pin 1 "вход": DD1_AI4)
	(* Не смотрим конкретную ошибку, / определяем,что вход неисправен без расшифровки. *)
	#113 DD1_AI4_QE0102:DECODE_FLOAT(VALUE: pin 1, DEF_VALUE: -)
	#114 NE(#113._ERR, 0)
	out 2 "авария" <= #114
	out 1 "выход" <= #113.OUT_VALUE
END_MACRO
#115 DD1_AI4_QE0102value <= #112.out 1
#116 DD1_AI4_error <= #112.out 2
#117 MACRO контроль аналогового входа DD1_AI5(pin 1 "вход": DD1_AI5)
	(* Не смотрим конкретную ошибку, / определяем,что вход неисправен без расшифровки. *)
	#118 DD1_AI5_FPK:DECODE_FLOAT(VALUE: pin 1, DEF_VALUE: -)
	#119 NE(#118._ERR, 0)
	out 2 "авария" <= #119
	out 1 "выход" <= #118.OUT_VALUE
END_MACRO
#120 DD1_AI5_FPKpressureValue <= #117.out 1
#121 DD1_AI5_error <= #117.out 2
#122 MACRO управление НД05.02 УПГ(pin 1 "вход расходомера в куб/час": DD1_AI1_FT0101value, pin 2 "max производительность НД в мл/мин": ND0502setMaxDosVal, pin 3 "задание дозирования в мл/куб": ND0502setKoefProp, pin 4 "режим:1 насос главный": ND0502regimeP1M, pin 5 "режим: 2 насос главный": ND0502regimeP2M, pin 6 "режим: по наработке": ND0502regimeByWT, pin 7 "режим: по кол-ву включений": ND0502regimeByC, pin 8 "авария 1 насоса": DD6_DI.0, pin 9 "авария 2 насоса": DD6_DI.1, pin 10 "сброс аварий": alarmReset, pin 11 "сброс счетчика включений 1 насоса": ND0502resetCountP1, pin 12 "сброс ссчетчика включений 2 насоса": ND0502resetCountP2, pin 13 "сброс наработки 1 насоса": ND0502resetWorkTimeP1, pin 14 "сброс наработки 2 насоса": ND0502resetWorkTimeP2)
	(* сигнал 4...20мА на НД05.02/02 *)
	(* сигнал 4...20мА на НД05.02/01 *)
	(* Если на входе SEL = TRUE, / то нижнее значение, / иначе - то,что посередине. *)
	#123 SEL(#130.pump1ON, 4, #124.outputValue)
	out 6 "выход 4...20мА насоса 1" <= #123
	#124 ND0502dosing:DosingPumpProportional(flowValue: pin 1, setMinPumpDosingValue: -, setMaxPumpDosingValue: pin 2, minOutputValue: -, maxOutputValue: -, setKoeffProportionality: pin 3, minFlowToStart: -)
	out 1 "ошибка блока дозирования" <= #124.dosingError
	#125 SEL(#130.pump2ON, 4, #124.outputValue)
	#126 linTrafND050201:LIN_TRAFO(IN: #125, IN_MIN: 4, IN_MAX: 20, OUT_MIN: 0, OUT_MAX: 1000)
	#127 REAL_TO_WORD(#126.OUT)
	out 7 "выход 4...20мА насоса 2" <= #127
	#128 ND0502regime:choosePumpRegime(start: #124.startDosingPump, pump1Main: pin 4, pump2Main: pin 5, byCounter: #129, byWorkTime: pin 6)
	out 2 "статус: 1 насос главный" <= #128.pump1MainActive
	out 3 "статус: 2 насос главный" <= #128.pump2MainActive
	out 4 "статус: по кол-ву включений" <= #128.byCounterActive
	#129 OR(pin 7, startInitializer)
	out 5 "статус: по наработке" <= #128.byWorkTimeActive
	#130 ND0502manager:TwoPumpManager(startStopPump1: #128.startPump1, startStopPump2: #128.startPump2, alarmPump1: #131, alarmPump2: #132, alarmReset: pin 10, counterStart: #128.startByCounter, Pump1ResetCounter: pin 11, Pump2ResetCounter: pin 12, ValueToResetCounter: -, workTimeStart: #128.startByWorkTime, workTimePump1Reset: pin 13, workTimePump2Reset: pin 14)
	out 12 "сигнал на включение насоса 1" <= #130.pump1ON
	#131 NOT(pin 8)
	out 13 "сигнал на включение насоса 2" <= #130.pump2ON
	out 8 "счетчик включений насоса 1" <= #130.counterPump1
	#132 NOT(pin 9)
	out 9 "счетчик включений насоса 2" <= #130.counterPump2
	out 10 "счетчик наработки насоса 1" <= #130.currentWorkTimePump1
	out 11 "счетчик наработки насоса 2" <= #130.currentWorkTimePump2
END_MACRO
#133 ND0502dosingError <= #122.out 1
#134 ND0502statRegimeP1M <= #122.out 2
#135 ND0502statRegimeP2M <= #122.out 3
#136 ND0502statRegimeByC <= #122.out 4
#137 ND0502statRegimeByWT <= #122.out 5
#138 DD1_AO3 <= #122.out 6
#139 DD10_AO0 <= #122.out 7
#140 ND0502counterP1 <= #122.out 8
#141 ND0502counterP2 <= #122.out 9
#142 ND0502workTimeP1 <= #122.out 10
#143 ND0502workTimeP2 <= #122.out 11
#144 DD4_DO.4 <= #122.out 12
#145 DD4_DO.5 <= #122.out 13
#146 AND(DD2_DO.1, DD5_DI.4)
#147 N0105statStartedP1 <= #146
#148 AND(DD5_DI.4, DD2_DO.2)
#149 N0105statStartedP2 <= #148
#150 MACRO Наполнение РЧВ02.03 (заслонка ЗДЭ02.25)(pin 1 "LS02.02раб.верх.уровень РЧВ": DD6_DI.14, pin 2 "LSA02.01 Перелив РЧВ": DD6_DI.13, pin 3 "статус ЗДЭ02.25 открыт": DD9_DI.0, pin 4 "статус ЗДЭ02.25 закрыт": DD9_DI.1, pin 5 "сброс аварий": alarmReset, pin 6 "время на открытие/закрытие": timeToOpenCloseValve)
	#151 OR(testZDE0225, pin 1)
	#152 NOT(pin 1)
	#153 ZDE0225:SimpleValve(inputOpen: #151, inputClose: #154, statusOpen: pin 3, statusClose: pin 4, reset: pin 5, timeToOpenClose: pin 6)
	out 1 "выход на открытие ЗДЭ02.25" <= #153.outputOpen
	#154 OR(#152, #155)
	out 2 "выход на закрытие ЗДЭ02.25" <= #153.outputClose
	out 3 "авария на открытие ЗДЭ02.25" <= #153.errorToOpen
	#155 NOT(pin 2)
	out 4 "авария на закрытие ЗДЭ02.25" <= #153.errorToClose
END_MACRO
#156 DD4_DO.0 <= #150.out 1
#157 DD4_DO.1 <= #150.out 2
#158 ZDE0225errorToOpen <= #150.out 3
#159 ZDE0225errorToClose <= #150.out 4
#160 MACRO управление Н02.04 (подача из РЧВ)(pin 1 "промывка ФС02.01/01": DD6_DI.20, pin 2 "промывка ФС02.01/02": DD6_DI.22, pin 3 "промывка ФС02.01/03": DD6_DI.24, pin 4 "промывка ФС02.01/04": DD6_DI.26, pin 5 "промывка ФС02.01/05": DD6_DI.28, pin 6 "промывка ФС02.01/06": DD6_DI.30, pin 7 "промывка ФС02.02/01": DD7_DI.0, pin 8 "промывка ФС02.02/02": DD7_DI.2, pin 9 "промывка ФС02.02/03": DD7_DI.4, pin 10 "промывка ФС02.02/04": DD7_DI.6, pin 11 "промывка ФС02.02/05": DD7_DI.8, pin 12 "промывка ФС02.02/06": DD7_DI.10, pin 13 "открыт КЭМ05.01": DD1_DI11, pin 14 "открыт КЭМ06.01": DD1_DI10, pin 15 "открыт КЭМ07.01": DD1_DI9, pin 16 "открыт КЭМ08.01": DD1_DI8, pin 17 "сухой ход Н02.04 (0=сух.ход)": DD5_DI.11, pin 18 "выбрать режим: Н02.04/01 - главный": N0204regimeP1M, pin 19 "выбрать режим: Н02.04/02 - главный": N0204regimeP2M, pin 20 "выбрать режим: по кол-ву включений": N0204regimeByC, pin 21 "выбрать режим: по наработке": N0204regimeWT, pin 22 "авария Н02.04/01 (0=авария)": DD5_DI.7, pin 23 "авария Н02.04/02 (0=авария)": DD5_DI.8, pin 24 "сброс аварий": alarmReset, pin 25 "сброс счетчика включений Н02.04/01": N0204resetCountP1, pin 26 "сброс счетчика включений Н02.04/02": N0204resetCountP2, pin 27 "сброс счетчика наработки Н02.04/01": N0204resetWorkTimeP1, pin 28 "сброс счетчика наработки Н02.04/02": N0204resetWorkTimeP2)
	(* Проверка, что фильтры 1 / ступени в регенерации (промывке) *)
	(* Проверка, что фильтры 2 / ступени в регенерации (промывке) *)
	(* Удержание сигнала на выключение насосов для / гарантированного сброса самоподхвата реле. *)
	(* Контроль открытия хотя бы одного из клапанов КЭМ *)
	(* сброс самоподхвата реле *)
	(* Защита от сухого хода Н02.04 / (LS02.03) 0=сух.ход *)
	#161 OR(pin 1, pin 2, pin 3, pin 4, pin 5, pin 6)
	#162 OR(#161, #163, #164)
	#163 OR(pin 7, pin 8, pin 9, pin 10, pin 11, pin 12)
	#164 OR(pin 13, pin 14, pin 15, pin 16)
	#165 N020401fTrigStop:F_TRIG(CLK: #172.pump1ON)
	#166 AND(#162, pin 17)
	#167 OR(#165.Q, #170.Q)
	#168 N0204stop:TOF(IN: #167, PT: T#1s)
	out 5 "стоп Н02.04" <= #168.Q
	#169 N0204chooseRegime:choosePumpRegime(start: #166, pump1Main: pin 18, pump2Main: pin 19, byCounter: #171, byWorkTime: pin 21)
	out 1 "выбран режим Н02.04/01 = главный" <= #169.pump1MainActive
	#170 N020402fTrigStop:F_TRIG(CLK: #172.pump2ON)
	out 2 "выбран режим Н02.04/02 = главный" <= #169.pump2MainActive
	out 3 "выбран режим по кол-ву включений" <= #169.byCounterActive
	#171 OR(pin 20, startInitializer)
	out 4 "выбран режим по наработке" <= #169.byWorkTimeActive
	#172 N0204manager:TwoPumpManager(startStopPump1: #169.startPump1, startStopPump2: #169.startPump2, alarmPump1: NOT pin 22, alarmPump2: NOT pin 23, alarmReset: pin 24, counterStart: #169.startByCounter, Pump1ResetCounter: pin 25, Pump2ResetCounter: pin 26, ValueToResetCounter: -, workTimeStart: #169.startByWorkTime, workTimePump1Reset: pin 27, workTimePump2Reset: pin 28)
	out 6 "пуск Н02.04/01" <= #172.pump1ON
	out 7 "пуск Н02.04/02" <= #172.pump2ON
	out 8 "счетчик включений Н02.04/01" <= #172.counterPump1
	out 9 "счетчик включений Н02.04/02" <= #172.counterPump2
	out 10 "счетчик наработки Н02.04/01" <= #172.currentWorkTimePump1
	out 11 "счетчик наработки Н02.04/02" <= #172.currentWorkTimePump2
END_MACRO
#173 N0204statRegimeP1M <= #160.out 1
#174 N0204statRegimeP2M <= #160.out 2
#175 N0204statRegimeByC <= #160.out 3
#176 N0204statRegimeWT <= #160.out 4
#177 DD4_DO.14 <= #160.out 5
#178 DD1_DO1 <= #160.out 6
#179 DD1_DO2 <= #160.out 7
#180 N0204counterP1 <= #160.out 8
#181 N0204counterP2 <= #160.out 9
#182 N0204workTimeP1 <= #160.out 10
#183 N0204workTimeP2 <= #160.out 11
#184 MACRO управление НД06.02 УПК(pin 1 "вход расходомера в куб/час": DD1_AI2_FT0102value, pin 2 "max производительность НД в мл/мин": ND0602setMaxDosVal, pin 3 "задание дозирования в мл/куб": ND0602setKoefProp, pin 4 "режим:1 насос главный": ND0602regimeP1M, pin 5 "режим: 2 насос главный": ND0602regimeP2M, pin 6 "режим: по наработке": ND0602regimeByWT, pin 7 "режим: по кол-ву включений": ND0602regimeByC, pin 8 "авария 1 насоса": DD6_DI.2, pin 9 "авария 2 насоса": DD6_DI.3, pin 10 "сброс аварий": alarmReset, pin 11 "сброс счетчика включений 1 насоса": ND0602resetCountP1, pin 12 "сброс ссчетчика включений 2 насоса": ND0602resetCountP2, pin 13 "сброс наработки 1 насоса": ND0602resetWorkTimeP1, pin 14 "сброс наработки 2 насоса": ND0602resetWorkTimeP2)
	(* сигнал 4...20мА на НД06.02/02 *)
	(* сигнал 4...20мА на НД06.02/01 *)
	(* Если на входе SEL = TRUE, / то нижнее значение, / иначе - то,что посередине. *)
	#185 SEL(#194.pump1ON, 4, #188.outputValue)
	#186 linTraf060201:LIN_TRAFO(IN: #185, IN_MIN: 4, IN_MAX: 20, OUT_MIN: 0, OUT_MAX: 1000)
	#187 REAL_TO_WORD(#186.OUT)
	out 6 "выход 4...20мА насоса 1" <= #187
	#188 ND0602dosing:DosingPumpProportional(flowValue: pin 1, setMinPumpDosingValue: -, setMaxPumpDosingValue: pin 2, minOutputValue: -, maxOutputValue: -, setKoeffProportionality: pin 3, minFlowToStart: -)
	out 1 "ошибка блока дозирования" <= #188.dosingError
	#189 SEL(#194.pump2ON, 4, #188.outputValue)
	#190 linTraf060202:LIN_TRAFO(IN: #189, IN_MIN: 4, IN_MAX: 20, OUT_MIN: 0, OUT_MAX: 1000)
	#191 REAL_TO_WORD(#190.OUT)
	out 7 "выход 4...20мА насоса 2" <= #191
	#192 ND0602regime:choosePumpRegime(start: #188.startDosingPump, pump1Main: pin 4, pump2Main: pin 5, byCounter: #193, byWorkTime: pin 6)
	out 2 "статус: 1 насос главный" <= #192.pump1MainActive
	out 3 "статус: 2 насос главный" <= #192.pump2MainActive
	out 4 "статус: по кол-ву включений" <= #192.byCounterActive
	#193 OR(pin 7, startInitializer)
	out 5 "статус: по наработке" <= #192.byWorkTimeActive
	#194 ND0602manager:TwoPumpManager(startStopPump1: #192.startPump1, startStopPump2: #192.startPump2, alarmPump1: #195, alarmPump2: #196, alarmReset: pin 10, counterStart: #192.startByCounter, Pump1ResetCounter: pin 11, Pump2ResetCounter: pin 12, ValueToResetCounter: -, workTimeStart: #192.startByWorkTime, workTimePump1Reset: pin 13, workTimePump2Reset: pin 14)
	out 12 "сигнал на включение насоса 1" <= #194.pump1ON
	#195 NOT(pin 8)
	out 13 "сигнал на включение насоса 2" <= #194.pump2ON
	out 8 "счетчик включений насоса 1" <= #194.counterPump1
	#196 NOT(pin 9)
	out 9 "счетчик включений насоса 2" <= #194.counterPump2
	out 10 "счетчик наработки насоса 1" <= #194.currentWorkTimePump1
	out 11 "счетчик наработки насоса 2" <= #194.currentWorkTimePump2
END_MACRO
#197 ND0602dosingError <= #184.out 1
#198 ND0602statRegimeP1M <= #184.out 2
#199 ND0602statRegimeP2M <= #184.out 3
#200 ND0602statRegimeByC <= #184.out 4
#201 ND0602statRegimeByWT <= #184.out 5
#202 DD10_AO1 <= #184.out 6
#203 DD10_AO2 <= #184.out 7
#204 ND0602counterP1 <= #184.out 8
#205 ND0602counterP2 <= #184.out 9
#206 ND0602workTimeP1 <= #184.out 10
#207 ND0602workTimeP2 <= #184.out 11
#208 DD4_DO.6 <= #184.out 12
#209 DD4_DO.7 <= #184.out 13
#210 OR(errorToOpenZDE0301, errorToCloseZDE0301, errorToOpenZDE0302, errorToCloseZDE0302)
#211 OR(DD5_DI.27, #210)
#212 OR(#210, DD5_DI.29)
#213 MACRO Работа УФО03.01(pin 1 "Работа УФО03.01/01": statusUFO030101started, pin 2 "Работа УФО03.01/02": statusUFO030102started, pin 3 "Значение расхода от FT01.02": DD1_AI2_FT0102value, pin 4 "мин.допустимый расход для насосов Н01.05": N0105minFlow, pin 5 "Задержка включения УФО на создание потока": UFO0301startDelayTime, pin 6 "выбор режим: УФО03.01/01 главное": UFO0301regimeP1M, pin 7 "выбор режим: УФО03.01/02 главное": UFO0301regimeP2M, pin 8 "выбор режим: по кол-ву включений": UFO0301regimeByC, pin 9 "выбор режим: по наработке": UFO0301regimeWT, pin 10 "авария УФО03.01/01": #211, pin 11 "авария УФО03.01/02": #212, pin 12 "сброс аварий": alarmReset, pin 13 "сброс счетчика включений УФО03.01/01": UFO0301resetCountP1, pin 14 "сброс счетчика включений УФО03.01/02": UFO0301resetCountP2, pin 15 "сброс счетчика наработки УФО03.01/01": UFO0301resetWorkTimeP1, pin 16 "сброс счетчика наработки УФО03.01/02": UFO0301resetWorkTimeP2)
	(* Контроль, если УФО включили вручную, / а потока при этом нет. *)
	(* Для подачи предостережения на пульте / оператора (при необходимости), а также / сигнализации лампой АВАРИЯ. *)
	(* Задержка старта УФО *)
	(* Включаем УФО, если расходомер показывает расход больше, / чем заданный как минимально допустимый для работы насосов Н01.05. *)
	#214 OR(pin 1, pin 2)
	#215 AND(#214, #216)
	out 1 "УФО вкл без потока" <= #215
	#216 NOT(#218.Q)
	#217 GE(pin 3, pin 4)
	#218 UFO0301startDelay:TON(IN: #217, PT: pin 5)
	#219 UFO0301regimeManager:choosePumpRegime(start: #218.Q, pump1Main: pin 6, pump2Main: pin 7, byCounter: #220, byWorkTime: pin 9)
	out 2 "активен режим - главное УФО 03.01/01" <= #219.pump1MainActive
	out 3 "активен режим - главное УФО 03.01/02" <= #219.pump2MainActive
	out 4 "активен режим - по кол-ву включений" <= #219.byCounterActive
	#220 OR(startInitializer, pin 8)
	out 5 "активен режим - по наработке" <= #219.byWorkTimeActive
	#221 UFO0301manager:TwoPumpManager(startStopPump1: #219.startPump1, startStopPump2: #219.startPump2, alarmPump1: pin 10, alarmPump2: pin 11, alarmReset: pin 12, counterStart: #219.startByCounter, Pump1ResetCounter: pin 13, Pump2ResetCounter: pin 14, ValueToResetCounter: -, workTimeStart: #219.startByWorkTime, workTimePump1Reset: pin 15, workTimePump2Reset: pin 16)
	out 6 "авт. пуск УФО03.01/01" <= #221.pump1ON
	out 7 "авт. пуск УФО03.01/02" <= #221.pump2ON
	out 8 "счетчик включений УФО03.01/01" <= #221.counterPump1
	out 9 "счетчик включений УФО03.01/02" <= #221.counterPump2
	out 10 "счетчик наработки УФО03.01/01" <= #221.currentWorkTimePump1
	out 11 "счетчик наработки УФО03.01/02" <= #221.currentWorkTimePump2
END_MACRO
#222 UFO0301noFlowAttention <= #213.out 1
#223 UFO0301statRegimeP1M <= #213.out 2
#224 UFO0301statRegimeP2M <= #213.out 3
#225 UFO0301statRegimeByC <= #213.out 4
#226 UFO0301statRegimeWT <= #213.out 5
#227 UFO0301counterP1 <= #213.out 8
#228 UFO0301counterP2 <= #213.out 9
#229 UFO0301workTimeP1 <= #213.out 10
#230 UFO0301workTimeP2 <= #213.out 11
#231 MACRO работа задвижек перед УФО и автом.пуск(pin 1 "сигнал на пуск УФО03.01/01": #213.out 6, pin 2 "сигнал на пуск УФО03.01/02": #213.out 7)
	(* авт.стопУФО03.01/02 *)
	(* авт.стопУФО03.01/01 *)
	(* авт.пускУФО03.01/02 *)
	(* авт.пускУФО03.01/01 *)
	(* 1 = тест задвижек ЗДЭ / 0 = возможность автом.пуска УФО *)
	(* 1 = открыть ЗДЭ03.01 / 0 = закрыть ЗДЭ03.01 *)
	(* 1 = открыть ЗДЭ03.02 / 0 = закрыть ЗДЭ03.02 *)
	#232 NOT(testZDE03)
	#233 NOT(testZDE03)
	#234 UFO030101startTrig:R_TRIG(CLK: #236)
	#235 UFO030101start <= #234.Q
	#236 AND(#232, #239, DD1_DI12)
	#237 UFO030101stopTrig:F_TRIG(CLK: #236)
	#238 UFO030101stop <= #237.Q
	#239 SEL(testZDE03, pin 1, manualZDE0301)
	#240 ZDE0301:SimpleValve(inputOpen: #239, inputClose: NOT #239, statusOpen: DD1_DI12, statusClose: DD1_DI13, reset: alarmReset, timeToOpenClose: timeToOpenCloseValve)
	#241 DD4_DO.16 <= #240.outputOpen
	#242 DD4_DO.17 <= #240.outputClose
	#243 errorToOpenZDE0301 <= #240.errorToOpen
	#244 errorToCloseZDE0301 <= #240.errorToClose
	#245 UFO030102startTrig:R_TRIG(CLK: #247)
	#246 UFO030102start <= #245.Q
	#247 AND(#233, #250, DD1_DI14)
	#248 UFO030102stopTrig:F_TRIG(CLK: #247)
	#249 UFO030102stop <= #248.Q
	#250 SEL(testZDE03, pin 2, manualZDE0302)
	#251 ZDE0302:SimpleValve(inputOpen: #250, inputClose: NOT #250, statusOpen: DD1_DI14, statusClose: DD1_DI15, reset: alarmReset, timeToOpenClose: timeToOpenCloseValve)
	#252 DD4_DO.18 <= #251.outputOpen
	#253 DD4_DO.19 <= #251.outputClose
	#254 errorToOpenZDE0302 <= #251.errorToOpen
	#255 errorToCloseZDE0302 <= #251.errorToClose
END_MACRO
#256 MACRO управление НД06.03 УПК(pin 1 "вход расходомера в куб/час": DD1_AI1_FT0101value, pin 2 "max производительность НД в мл/мин": ND0603setMaxDosVal, pin 3 "задание дозирования в мл/куб": ND0603setKoefProp, pin 4 "режим:1 насос главный": ND0603regimeP1M, pin 5 "режим: 2 насос главный": ND0603regimeP2M, pin 6 "режим: по наработке": ND0603regimeByWT, pin 7 "режим: по кол-ву включений": ND0603regimeByC, pin 8 "авария 1 насоса": DD6_DI.4, pin 9 "авария 2 насоса": DD6_DI.5, pin 10 "сброс аварий": alarmReset, pin 11 "сброс счетчика включений 1 насоса": ND0603resetCountP1, pin 12 "сброс ссчетчика включений 2 насоса": ND0603resetCountP2, pin 13 "сброс наработки 1 насоса": ND0603resetWorkTimeP1, pin 14 "сброс наработки 2 насоса": ND0603resetWorkTimeP2)
	(* сигнал 4...20мА на НД06.03/02 *)
	(* сигнал 4...20мА на НД06.03/01 *)
	(* Если на входе SEL = TRUE, / то нижнее значение, / иначе - то,что посередине. *)
	#257 SEL(#266.pump1ON, 4, #260.outputValue)
	#258 linTraf060301:LIN_TRAFO(IN: #257, IN_MIN: 4, IN_MAX: 20, OUT_MIN: 0, OUT_MAX: 1000)
	#259 REAL_TO_WORD(#258.OUT)
	out 6 "выход 4...20мА насоса 1" <= #259
	#260 ND0603dosing:DosingPumpProportional(flowValue: pin 1, setMinPumpDosingValue: -, setMaxPumpDosingValue: pin 2, minOutputValue: -, maxOutputValue: -, setKoeffProportionality: pin 3, minFlowToStart: -)
	out 1 "ошибка блока дозирования" <= #260.dosingError
	#261 SEL(#266.pump2ON, 4, #260.outputValue)
	#262 linTraf060302:LIN_TRAFO(IN: #261, IN_MIN: 4, IN_MAX: 20, OUT_MIN: 0, OUT_MAX: 1000)
	#263 REAL_TO_WORD(#262.OUT)
	out 7 "выход 4...20мА насоса 2" <= #263
	#264 ND0603regime:choosePumpRegime(start: #260.startDosingPump, pump1Main: pin 4, pump2Main: pin 5, byCounter: #265, byWorkTime: pin 6)
	out 2 "статус: 1 насос главный" <= #264.pump1MainActive
	out 3 "статус: 2 насос главный" <= #264.pump2MainActive
	out 4 "статус: по кол-ву включений" <= #264.byCounterActive
	#265 OR(pin 7, startInitializer)
	out 5 "статус: по наработке" <= #264.byWorkTimeActive
	#266 ND0603manager:TwoPumpManager(startStopPump1: #264.startPump1, startStopPump2: #264.startPump2, alarmPump1: #267, alarmPump2: #268, alarmReset: pin 10, counterStart: #264.startByCounter, Pump1ResetCounter: pin 11, Pump2ResetCounter: pin 12, ValueToResetCounter: -, workTimeStart: #264.startByWorkTime, workTimePump1Reset: pin 13, workTimePump2Reset: pin 14)
	out 12 "сигнал на включение насоса 1" <= #266.pump1ON
	#267 NOT(pin 8)
	out 13 "сигнал на включение насоса 2" <= #266.pump2ON
	out 8 "счетчик включений насоса 1" <= #266.counterPump1
	#268 NOT(pin 9)
	out 9 "счетчик включений насоса 2" <= #266.counterPump2
	out 10 "счетчик наработки насоса 1" <= #266.currentWorkTimePump1
	out 11 "счетчик наработки насоса 2" <= #266.currentWorkTimePump2
END_MACRO
#269 ND0603dosingError <= #256.out 1
#270 ND0603statRegimeP1M <= #256.out 2
#271 ND0603statRegimeP2M <= #256.out 3
#272 ND0603statRegimeByC <= #256.out 4
#273 ND0603statRegimeByWT <= #256.out 5
#274 DD10_AO3 <= #256.out 6
#275 DD10_AO4 <= #256.out 7
#276 ND0603counterP1 <= #256.out 8
#277 ND0603counterP2 <= #256.out 9
#278 ND0603workTimeP1 <= #256.out 10
#279 ND0603workTimeP2 <= #256.out 11
#280 DD4_DO.8 <= #256.out 12
#281 DD4_DO.9 <= #256.out 13
#282 MACRO управление Н04.04 (дренажные)(pin 1 "защита от сухого хода Н04.04": DD5_DI.18, pin 2 "автоматич.пускН04.04": DD5_DI.19, pin 3 "режим Н04.04/01 главный": N0404regimeP1M, pin 4 "режим Н04.04/02 главный": N0404regimeP2M, pin 5 "режим по кол-ву включений": N0404regimeByC, pin 6 "режим по наработке": N0404regimeWT, pin 7 "авария Н04.04/01": DD5_DI.15, pin 8 "авария Н04.04/02": DD5_DI.14, pin 9 "сброс аварий": alarmReset, pin 10 "сброс счетчика включений Н04.04/01": N0404resetCountP1, pin 11 "сброс счетчика включений Н04.04/02": N0404resetCountP2, pin 12 "сброс счетчика наработки Н04.04/01": N0404resetWorkTimeP1, pin 13 "сброс счетчика наработки Н04.04/02": N0404resetWorkTimeP2)
	(* сбрасывает самоподхват пускового реле *)
	(* Излишняя перестраховка по сухому ходу, / на уровне реле уже все отрабатывается. *)
	(* насосы имеют электрическую блокировку / от одновременного включения *)
	(* от поплавка *)
	(* сухой ход Н04.04 / 0=защита *)
	(* 0=авария *)
	#283 NOT(pin 1)
	out 1 "стоп Н04.04" <= #283
	#284 AND(pin 1, pin 2)
	#285 N0401choosePumpRegime:choosePumpRegime(start: #284, pump1Main: pin 3, pump2Main: pin 4, byCounter: #286, byWorkTime: pin 6)
	out 2 "выбран режим: Н04.04/01 главный" <= #285.pump1MainActive
	out 3 "выбран режим: Н04.04/02 главный" <= #285.pump2MainActive
	out 4 "выбран режим: по кол-ву включений" <= #285.byCounterActive
	#286 OR(startInitializer, pin 5)
	out 5 "выбран режим: по наработке" <= #285.byWorkTimeActive
	#287 N0404twoPumpManager:TwoPumpManager(startStopPump1: #285.startPump1, startStopPump2: #285.startPump2, alarmPump1: #288, alarmPump2: #289, alarmReset: pin 9, counterStart: #285.startByCounter, Pump1ResetCounter: pin 10, Pump2ResetCounter: pin 11, ValueToResetCounter: -, workTimeStart: #285.startByWorkTime, workTimePump1Reset: pin 12, workTimePump2Reset: pin 13)
	out 6 "пуск Н04.04/01" <= #287.pump1ON
	#288 NOT(pin 7)
	out 7 "пуск Н04.04/02" <= #287.pump2ON
	out 8 "счетчик кол-ва включений Н04.04/01" <= #287.counterPump1
	#289 NOT(pin 8)
	out 9 "счетчик кол-ва включений Н04.04/02" <= #287.counterPump2
	out 10 "счетчик времени наработки Н04.04/01" <= #287.currentWorkTimePump1
	out 11 "счетчик времени наработки Н04.04/02" <= #287.currentWorkTimePump2
END_MACRO
#290 DD4_DO.15 <= #282.out 1
#291 N0404statRegimeP1M <= #282.out 2
#292 N0404statRegimeP2M <= #282.out 3
#293 N0404statRegimeByC <= #282.out 4
#294 N0404statRegimeWT <= #282.out 5
#295 DD1_DO5 <= #282.out 6
#296 DD1_DO6 <= #282.out 7
#297 N0404counterP1 <= #282.out 8
#298 N0404counterP2 <= #282.out 9
#299 N0404workTimeP1 <= #282.out 10
#300 N0404workTimeP2 <= #282.out 11
#301 MACRO управление НД07.03 УПЩ (поддержка рН, ПИД-регулятор)(pin 1 "вход рН-метра QE01.01": DD1_AI3_QE0101value, pin 2 "уставка рН": ND0703pHsetValue, pin 3 "режим:1 насос главный": ND0703regimeP1M, pin 4 "режим: 2 насос главный": ND0703regimeP2M, pin 5 "режим: по наработке": ND0703regimeByWT, pin 6 "режим: по кол-ву включений": ND0703regimeByC, pin 7 "авария 1 насоса": DD6_DI.6, pin 8 "авария 2 насоса": DD6_DI.7, pin 9 "сброс аварий": alarmReset, pin 10 "сброс счетчика включений 1 насоса": ND0703resetCountP1, pin 11 "сброс счетчика включений 2 насоса": ND0703resetCountP2, pin 12 "сброс наработки 1 насоса": ND0703resetWorkTimeP1, pin 13 "сброс наработки 2 насоса": ND0703resetWorkTimeP2, pin 14 "ручное управл.выходом Y (4...20мА)": ND0703YoutManual, pin 15 "1=ручное/0=автомат.управл.": ND0703YmanAuto, pin 16 "вход расходомера FT01.01 (куб.м/час)": DD1_AI1_FT0101value, pin 17 "коэфф.I": ND0703koeffI, pin 18 "коэфф.D": ND0703koeffD, pin 19 "коэфф.Р": ND0703koeffP)
	(* сигнал 4...20мА на НД07.03/02 *)
	(* сигнал 4...20мА на НД07.03/01 *)
	(* Если на входе SEL = TRUE, / то нижнее значение, / иначе - то,что посередине. *)
	(* min расход в кубометрах в час / для неачала дозирования. *)
	#302 ND0703pidReg:PID(ACTUAL: pin 1, SET_POINT: pin 2, KP: pin 19, TN: pin 17, TV: pin 18, Y_MANUAL: pin 14, Y_OFFSET: 12, Y_MIN: 0, Y_MAX: 1000, MANUAL: pin 15, RESET: #302.OVERFLOW)
	#303 SEL(#310.pump1ON, 0, #302.Y)
	#304 REAL_TO_WORD(#303)
	out 5 "выход 4...20мА насоса 1" <= #304
	#305 SEL(#310.pump2ON, 0, #302.Y)
	#306 REAL_TO_WORD(#305)
	out 6 "выход 4...20мА насоса 2" <= #306
	#307 GE(pin 16, 10)
	#308 ND0703regime:choosePumpRegime(start: #307, pump1Main: pin 3, pump2Main: pin 4, byCounter: #309, byWorkTime: pin 5)
	out 1 "статус: 1 насос главный" <= #308.pump1MainActive
	out 2 "статус: 2 насос главный" <= #308.pump2MainActive
	out 3 "статус: по кол-ву включений" <= #308.byCounterActive
	out 4 "статус: по наработке" <= #308.byWorkTimeActive
	#309 OR(pin 6, startInitializer)
	#310 ND0703manager:TwoPumpManager(startStopPump1: #308.startPump1, startStopPump2: #308.startPump2, alarmPump1: #311, alarmPump2: #312, alarmReset: pin 9, counterStart: #308.startByCounter, Pump1ResetCounter: pin 10, Pump2ResetCounter: pin 11, ValueToResetCounter: -, workTimeStart: #308.startByWorkTime, workTimePump1Reset: pin 12, workTimePump2Reset: pin 13)
	out 11 "сигнал на включение насоса 1" <= #310.pump1ON
	#311 NOT(pin 7)
	out 12 "сигнал на включение насоса 2" <= #310.pump2ON
	out 7 "счетчик включений насоса 1" <= #310.counterPump1
	#312 NOT(pin 8)
	out 8 "счетчик включений насоса 2" <= #310.counterPump2
	out 9 "счетчик наработки насоса 1" <= #310.currentWorkTimePump1
	out 10 "счетчик наработки насоса 2" <= #310.currentWorkTimePump2
END_MACRO
#313 ND0703statRegimeP1M <= #301.out 1
#314 ND0703statRegimeP2M <= #301.out 2
#315 ND0703statRegimeByC <= #301.out 3
#316 ND0703statRegimeByWT <= #301.out 4
#317 DD10_AO5 <= #301.out 5
#318 DD10_AO6 <= #301.out 6
#319 ND0703counterP1 <= #301.out 7
#320 ND0703counterP2 <= #301.out 8
#321 ND0703workTimeP1 <= #301.out 9
#322 ND0703workTimeP2 <= #301.out 10
#323 DD4_DO.10 <= #301.out 11
#324 DD4_DO.11 <= #301.out 12
#325 MACRO импульсный счетчик FQS0301(pin 1 "вход от счетчика": DD6_DI.19, pin 2 "вес импульса счетчика": FQS0301impulsValue, pin 3 "сброс счетчика": FQS0301reset, pin 4 "величина коррекции счетчика": FQS0301correction, pin 5 "прибавить коррекцию": FQS0301addCorrection, pin 6 "вычесть коррекцию": FQS0301deleteCorrection)
	(* сброс показаний счетчика *)
	(* значение в REAL (в какой-то момент начинает / отображаться в экспоненциальной форме) *)
	(* Если в результате коррекции накопленная сумма станет меньше нуля, то она принудительно станет равна нулю. *)
	(* коррекция показаний счетчика. *)
	(* число, коорое будем прибавлять или / вычитать из накопленной суммы стоков. *)
	#326 FQS0301rTrig:R_TRIG(CLK: pin 1)
	#327 ADD(EN: #326.Q, FQS0301totalAmount, pin 2)
	out 1 "накопленная сумма стоков (REAL)" <= #327
	#328 FQS0301resetRtrig:R_TRIG(CLK: pin 3)
	#329 MOVE(EN: #328.Q, 0)
	#330 FQS0301totalAmount <= #329
	#331 FQS0301addCorrRtrig:R_TRIG(CLK: pin 5)
	#332 ADD(EN: #331.Q, FQS0301totalAmount, pin 4)
	#333 FQS0301totalAmount <= #332
	#334 FQS0301deleteCorrRtrig:R_TRIG(CLK: pin 6)
	#335 SUB(EN: #334.Q, FQS0301totalAmount, pin 4)
	#336 FQS0301totalAmount <= #335
	#337 LT(FQS0301totalAmount, 0)
	#338 MOVE(EN: #337, 0)
	#339 FQS0301totalAmount <= #338
END_MACRO
#340 FQS0301totalAmount <= #325.out 1
#341 MACRO управление НД08.03 УПФ(pin 1 "вход расходомера в куб/час": DD1_AI1_FT0101value, pin 2 "max производительность НД в мл/мин": ND0803setMaxDosVal, pin 3 "задание дозирования в мл/куб": ND0803setKoefProp, pin 4 "режим:1 насос главный": ND0803regimeP1M, pin 5 "режим: 2 насос главный": ND0803regimeP2M, pin 6 "режим: по наработке": ND0803regimeByWT, pin 7 "режим: по кол-ву включений": ND0803regimeByC, pin 8 "авария 1 насоса": DD5_DI.12, pin 9 "авария 2 насоса": DD5_DI.13, pin 10 "сброс аварий": alarmReset, pin 11 "сброс счетчика включений 1 насоса": ND0803resetCountP1, pin 12 "сброс ссчетчика включений 2 насоса": ND0803resetCountP2, pin 13 "сброс наработки 1 насоса": ND0803resetWorkTimeP1, pin 14 "сброс наработки 2 насоса": ND0803resetWorkTimeP2, pin 15 "сухой ход 1 насоса": DD1_DI6, pin 16 "сухой ход 2 насоса": DD1_DI7)
	(* сигнал 4...20мА на НД08.03/02 *)
	(* сигнал 4...20мА на НД08.03/01 *)
	(* Если на входе SEL = TRUE, / то нижнее значение, / иначе - то,что посередине. *)
	#342 SEL(#351.pump1ON, 0, #343.outputValue)
	out 6 "выход 4...20мА насоса 1" <= #342
	#343 ND0803dosing:DosingPumpProportional(flowValue: pin 1, setMinPumpDosingValue: -, setMaxPumpDosingValue: pin 2, minOutputValue: -, maxOutputValue: -, setKoeffProportionality: pin 3, minFlowToStart: -)
	out 1 "ошибка блока дозирования" <= #343.dosingError
	#344 SEL(#351.pump2ON, 0, #343.outputValue)
	out 7 "выход 4...20мА насоса 2" <= #344
	#345 ND0803regime:choosePumpRegime(start: #343.startDosingPump, pump1Main: pin 4, pump2Main: pin 5, byCounter: #346, byWorkTime: pin 6)
	out 2 "статус: 1 насос главный" <= #345.pump1MainActive
	out 3 "статус: 2 насос главный" <= #345.pump2MainActive
	out 4 "статус: по кол-ву включений" <= #345.byCounterActive
	#346 OR(pin 7, startInitializer)
	out 5 "статус: по наработке" <= #345.byWorkTimeActive
	out 12 "сигнал на включение насоса 1" <= #351.pump1ON
	#347 NOT(pin 8)
	#348 OR(#347, pin 15)
	out 13 "сигнал на включение насоса 2" <= #351.pump2ON
	#349 NOT(pin 9)
	#350 OR(#349, pin 16)
	#351 ND0803manager:TwoPumpManager(startStopPump1: #345.startPump1, startStopPump2: #345.startPump2, alarmPump1: #348, alarmPump2: #350, alarmReset: pin 10, counterStart: #345.startByCounter, Pump1ResetCounter: pin 11, Pump2ResetCounter: pin 12, ValueToResetCounter: -, workTimeStart: #345.startByWorkTime, workTimePump1Reset: pin 13, workTimePump2Reset: pin 14)
	out 8 "счетчик включений насоса 1" <= #351.counterPump1
	out 9 "счетчик включений насоса 2" <= #351.counterPump2
	out 10 "счетчик наработки насоса 1" <= #351.currentWorkTimePump1
	out 11 "счетчик наработки насоса 2" <= #351.currentWorkTimePump2
END_MACRO
#352 ND0803dosingError <= #341.out 1
#353 ND0803statRegimeP1M <= #341.out 2
#354 ND0803statRegimeP2M <= #341.out 3
#355 ND0803statRegimeByC <= #341.out 4
#356 ND0803statRegimeByWT <= #341.out 5
#357 DD1_AO1 <= #341.out 6
#358 DD1_AO2 <= #341.out 7
#359 ND0803counterP1 <= #341.out 8
#360 ND0803counterP2 <= #341.out 9
#361 ND0803workTimeP1 <= #341.out 10
#362 ND0803workTimeP2 <= #341.out 11
#363 DD1_DO3 <= #341.out 12
#364 DD1_DO4 <= #341.out 13
#365 AND(DD1_DI5, DD1_DI4, DD6_DI.11)
#366 DD1_DO8 <= #365
#367 EQ(lastError, 0)
#368 alarmPLKnetworkDelay:TOF(IN: #367, PT: T#20s)
#369 NOT(#368.Q)
#370 alarmPLKnetwork <= #369
#371 MACRO управление НД08.04 УПФ(pin 1 "насос Н04.01 работает": DD7_DI.13, pin 2 "авария НД08.04": DD6_DI.16, pin 3 "уставкаНД08.04(0...100%)": ND0804doseValue)
	(* Преобразует сигнал 0...100 / пропорционально в 4...20мА *)
	#372 AND(pin 1, pin 2)
	out 1 "пуск/стоп НД08.04" <= #372
	#373 ND0804linearTransformator:LIN_TRAFO(IN: pin 3, IN_MIN: 0, IN_MAX: 100, OUT_MIN: 0, OUT_MAX: 1000)
	#374 REAL_TO_WORD(#373.OUT)
	out 2 "управление НД08.04 (4...20мА)" <= #374
	out 3 "ошибка блока дозирования" <= #373.ERROR
END_MACRO
#375 DD4_DO.12 <= #371.out 1
#376 DD10_AO7 <= #371.out 2
#377 ND0804dosingError <= #371.out 3
#378 NOT(DD6_DI.0)
#379 alarmND050201 <= #378
#380 NOT(DD6_DI.23)
#381 alarmFS020102 <= #380
#382 NOT(DD9_DI.14)
#383 alarmZDE0211power <= #382
#384 NOT(DD6_DI.1)
#385 alarmND050202 <= #384
#386 NOT(DD6_DI.25)
#387 alarmFS020103 <= #386
#388 NOT(DD9_DI.15)
#389 alarmZDE0212power <= #388
#390 NOT(DD6_DI.2)
#391 alarmND060201 <= #390
#392 NOT(DD6_DI.27)
#393 alarmFS020104 <= #392
#394 NOT(DD9_DI.16)
#395 alarmZDE0213power <= #394
#396 NOT(DD6_DI.3)
#397 alarmND060202 <= #396
#398 NOT(DD6_DI.29)
#399 alarmFS020105 <= #398
#400 NOT(DD9_DI.17)
#401 alarmZDE0214power <= #400
#402 MACRO контроль включения мешалок(pin 1 "работа НД06.02/01": DD4_DO.6, pin 2 "работа НД06.02/02": DD4_DO.7, pin 3 "работа НД06.03/01": DD4_DO.8, pin 4 "работа НД06.03/02": DD4_DO.9, pin 5 "работа мешалки М06.04": DD5_DI.21, pin 6 "работа НД07.03/01": DD4_DO.10, pin 7 "работа НД07.03/02": DD4_DO.11, pin 8 "работа мешалки М07.02": DD5_DI.23, pin 9 "работа НД08.03/01": DD1_DO3, pin 10 "работа НД08.03/02": DD1_DO4, pin 11 "работа НД08.04": DD4_DO.12, pin 12 "работа мешалки М08.02": DD5_DI.25)
	#403 OR(pin 1, pin 2, pin 3, pin 4)
	#404 AND(#403, #405)
	out 1 "дозирования при выключенной М06.04" <= #404
	#405 NOT(pin 5)
	#406 OR(pin 6, pin 7)
	#407 AND(#406, #408)
	out 2 "дозирования при выключенной М07.02" <= #407
	#408 NOT(pin 8)
	#409 OR(pin 9, pin 10, pin 11)
	#410 AND(#409, #411)
	out 3 "дозирования при выключенной М08.02" <= #410
	#411 NOT(pin 12)
END_MACRO
#412 M0604attention <= #402.out 1
#413 M0702attention <= #402.out 2
#414 M0802attention <= #402.out 3
#415 NOT(DD6_DI.4)
#416 alarmND060301 <= #415
#417 NOT(DD6_DI.31)
#418 alarmFS020106 <= #417
#419 NOT(DD9_DI.18)
#420 alarmZDE0215power <= #419
#421 NOT(DD6_DI.5)
#422 alarmND060302 <= #421
#423 NOT(DD7_DI.1)
#424 alarmFS020201 <= #423
#425 NOT(DD9_DI.19)
#426 alarmZDE0216power <= #425
#427 NOT(DD6_DI.6)
#428 alarmND070301 <= #427
#429 NOT(DD7_DI.3)
#430 alarmFS020202 <= #429
#431 NOT(DD9_DI.20)
#432 alarmZDE0217power <= #431
#433 NOT(DD6_DI.7)
#434 alarmND070302 <= #433
#435 NOT(DD7_DI.5)
#436 alarmFS020203 <= #435
#437 NOT(DD9_DI.21)
#438 alarmZDE0218power <= #437
#439 NOT(DD5_DI.12)
#440 alarmND080301 <= #439
#441 NOT(DD7_DI.7)
#442 alarmFS020204 <= #441
#443 NOT(DD9_DI.22)
#444 alarmZDE0219power <= #443
#445 NOT(DD5_DI.13)
#446 alarmND080302 <= #445
#447 NOT(DD7_DI.9)
#448 alarmFS020205 <= #447
#449 NOT(DD9_DI.23)
#450 alarmZDE0220power <= #449
#451 NOT(DD6_DI.16)
#452 alarmND0804 <= #451
#453 NOT(DD7_DI.11)
#454 alarmFS020206 <= #453
#455 NOT(DD9_DI.24)
#456 alarmZDE0221power <= #455
#457 NOT(DD6_DI.11)
#458 alarmOGM0104overload <= #457
#459 NOT(DD9_DI.4)
#460 alarmZDE0201power <= #459
#461 NOT(DD9_DI.25)
#462 alarmZDE0222power <= #461
#463 MACRO переменные для обмена с панелью()
	#464 MACRO PSW регистры на передачу в панель (отображение)()
		(* PSW регистры на передачу в панель (отображение) *)
		(* panFQS0301totalAmount - переменная отображена сразу на выходе соответствующего макроса (учет очищенных стоков). / Здесь не хранится. *)
		#465 panFT0101value <= DD1_AI1_FT0101value
		#466 panQE0101value <= DD1_AI3_QE0101value
		#467 panFT0102value <= DD1_AI2_FT0102value
		#468 panQE0102value <= DD1_AI4_QE0102value
		#469 panFPKpressureValue <= DD1_AI5_FPKpressureValue
		#470 panFQS0301total <= FQS0301totalAmount
		#471 panTemperature <= temperatureValue
		#472 MACRO Время наработки и кол-во включений агрегатов()
			#473 workTimeND050201:TimeFromWorkTime(input: ND0502workTimeP1)
			#474 panND050201workDays <= #473.days
			#475 panND050201workHours <= #473.hours
			#476 panND050201workMinutes <= #473.minutes
			#477 panND050201workSeconds <= #473.seconds
			#478 workTimeND050202:TimeFromWorkTime(input: ND0502workTimeP2)
			#479 panND050202workDays <= #478.days
			#480 panND050202workHours <= #478.hours
			#481 panND050202workMinutes <= #478.minutes
			#482 panND050202workSeconds <= #478.seconds
			#483 panND0502counterP1 <= ND0502counterP1
			#484 panND0502counterP2 <= ND0502counterP2
			#485 workTimeND060201:TimeFromWorkTime(input: ND0602workTimeP1)
			#486 panND060201workDays <= #485.days
			#487 panND060201workHours <= #485.hours
			#488 panND060201workMinutes <= #485.minutes
			#489 panND060201workSeconds <= #485.seconds
			#490 workTimeND060202:TimeFromWorkTime(input: ND0602workTimeP2)
			#491 panND060202workDays <= #490.days
			#492 panND060202workHours <= #490.hours
			#493 panND060202workMinutes <= #490.minutes
			#494 panND060202workSeconds <= #490.seconds
			#495 panND0602counterP1 <= ND0602counterP1
			#496 panND0602counterP2 <= ND0602counterP2
			#497 workTimeND060301:TimeFromWorkTime(input: ND0603workTimeP1)
			#498 panND060301workDays <= #497.days
			#499 panND060301workHours <= #497.hours
			#500 panND060301workMinutes <= #497.minutes
			#501 panND060301workSeconds <= #497.seconds
			#502 workTimeND060302:TimeFromWorkTime(input: ND0603workTimeP2)
			#503 panND060302workDays <= #502.days
			#504 panND060302workHours <= #502.hours
			#505 panND060302workMinutes <= #502.minutes
			#506 panND060302workSeconds <= #502.seconds
			#507 panND0603counterP1 <= ND0603counterP1
			#508 panND0603counterP2 <= ND0603counterP2
			#509 workTimeND070301:TimeFromWorkTime(input: ND0703workTimeP1)
			#510 panND070301workDays <= #509.days
			#511 panND070301workHours <= #509.hours
			#512 panND070301workMinutes <= #509.minutes
			#513 panND070301workSeconds <= #509.seconds
			#514 workTimeND070302:TimeFromWorkTime(input: ND0703workTimeP2)
			#515 panND070302workDays <= #514.days
			#516 panND070302workHours <= #514.hours
			#517 panND070302workMinutes <= #514.minutes
			#518 panND070302workSeconds <= #514.seconds
			#519 panND0703counterP1 <= ND0703counterP1
			#520 panND0703counterP2 <= ND0703counterP2
			#521 workTimeND080301:TimeFromWorkTime(input: ND0803workTimeP1)
			#522 panND080301workDays <= #521.days
			#523 panND080301workHours <= #521.hours
			#524 panND080301workMinutes <= #521.minutes
			#525 panND080301workSeconds <= #521.seconds
			#526 workTimeND080302:TimeFromWorkTime(input: ND0803workTimeP2)
			#527 panND080302workDays <= #526.days
			#528 panND080302workHours <= #526.hours
			#529 panND080302workMinutes <= #526.minutes
			#530 panND080302workSeconds <= #526.seconds
			#531 panND0803counterP1 <= ND0803counterP1
			#532 panND0803counterP2 <= ND0803counterP2
			#533 workTimeN010501:TimeFromWorkTime(input: N0105workTimeP1)
			#534 panN010501workDays <= #533.days
			#535 panN010501workHours <= #533.hours
			#536 panN010501workMinutes <= #533.minutes
			#537 panN010501workSeconds <= #533.seconds
			#538 workTimeN010502:TimeFromWorkTime(input: N0105workTimeP2)
			#539 panN010502workDays <= #538.days
			#540 panN010502workHours <= #538.hours
			#541 panN010502workMinutes <= #538.minutes
			#542 panN010502workSeconds <= #538.seconds
			#543 panN0105counterP1 <= N0105counterP1
			#544 panN0105counterP2 <= N0105counterP2
			#545 workTimeN020401:TimeFromWorkTime(input: N0204workTimeP1)
			#546 panN020401workDays <= #545.days
			#547 panN020401workHours <= #545.hours
			#548 panN020401workMinutes <= #545.minutes
			#549 panN020401workSeconds <= #545.seconds
			#550 workTimeN020402:TimeFromWorkTime(input: N0204workTimeP2)
			#551 panN020402workDays <= #550.days
			#552 panN020402workHours <= #550.hours
			#553 panN020402workMinutes <= #550.minutes
			#554 panN020402workSeconds <= #550.seconds
			#555 panN0204counterP1 <= N0204counterP1
			#556 panN0204counterP2 <= N0204counterP2
			#557 workTimeN040401:TimeFromWorkTime(input: N0404workTimeP1)
			#558 panN040401workDays <= #557.days
			#559 panN040401workHours <= #557.hours
			#560 panN040401workMinutes <= #557.minutes
			#561 panN040401workSeconds <= #557.seconds
			#562 workTimeN040402:TimeFromWorkTime(input: N0404workTimeP2)
			#563 panN040402workDays <= #562.days
			#564 panN040402workHours <= #562.hours
			#565 panN040402workMinutes <= #562.minutes
			#566 panN040402workSeconds <= #562.seconds
			#567 panN0404counterP1 <= N0404counterP1
			#568 panN0404counterP2 <= N0404counterP2
			#569 workTimeUFO030101:TimeFromWorkTime(input: UFO0301workTimeP1)
			#570 panUFO030101workDays <= #569.days
			#571 panUFO030101workHours <= #569.hours
			#572 panUFO030101workMinutes <= #569.minutes
			#573 panUFO030101workSeconds <= #569.seconds
			#574 workTimeUFO030102:TimeFromWorkTime(input: UFO0301workTimeP2)
			#575 panUFO030102workDays <= #574.days
			#576 panUFO030102workHours <= #574.hours
			#577 panUFO030102workMinutes <= #574.minutes
			#578 panUFO030102workSeconds <= #574.seconds
			#579 panUFO0301counterP1 <= UFO0301counterP1
			#580 panUFO0301counterP2 <= UFO0301counterP2
		END_MACRO
		#581 panVolumeToRegen <= volumeToRegen
	END_MACRO
	#582 MACRO PSB регистры на передачу в панель (отображение)()
		(* PSB регистры на передачу в панель (отображение) *)
		#583 MACRO 8 bit output module 1()
			#584 panStartND050201 <= DD4_DO.4
			#585 panStartND050202 <= DD4_DO.5
			#586 panStartND060201 <= DD4_DO.6
			#587 panStartND060202 <= DD4_DO.7
			#588 panStartND060301 <= DD4_DO.8
			#589 panStartND060302 <= DD4_DO.9
			#590 panStartM0604 <= DD5_DI.21
			#591 panStartND070301 <= DD4_DO.10
		END_MACRO
		#592 MACRO 8 bit output module 2()
			#593 panStartND070302 <= DD4_DO.11
			#594 panStartM0702 <= DD5_DI.23
			#595 panStartND080301 <= DD1_DO3
			#596 panStartND080302 <= DD1_DO4
			#597 panStartND0804 <= DD4_DO.12
			#598 panStartM0802 <= DD5_DI.25
			#599 panStartN020401 <= DD5_DI.9
			#600 panStartN020402 <= DD5_DI.10
		END_MACRO
		#601 MACRO 8 bit output module 3()
			#602 panStartN010501 <= N0105statStartedP1
			#603 panStartN010502 <= N0105statStartedP2
			#604 panCleanFS020101 <= DD6_DI.20
			#605 panCleanFS020102 <= DD6_DI.22
			#606 panCleanFS020103 <= DD6_DI.24
			#607 panCleanFS020104 <= DD6_DI.26
			#608 panCleanFS020105 <= DD6_DI.28
			#609 panCleanFS020106 <= DD6_DI.30
		END_MACRO
		#610 MACRO 8 bit output module 4()
			#611 panCleanFS020201 <= DD7_DI. 0
			#612 panCleanFS020202 <= DD7_DI. 2
			#613 panCleanFS020203 <= DD7_DI. 4
			#614 panCleanFS020204 <= DD7_DI. 6
			#615 panCleanFS020205 <= DD7_DI. 8
			#616 panCleanFS020206 <= DD7_DI. 10
			#617 panSludgeReady <= DD7_DI.15
			#618 panStartN0401 <= DD7_DI.13
		END_MACRO
		#619 MACRO 8 bit output module 5()
			#620 panKSHE0401open <= DD9_DI.2
			#621 panFPKready <= DD7_DI.12
			#622 panFPKneedToClean <= FPKneedToClean
			#623 panStartN040401 <= DD5_DI.16
			#624 panStartN040402 <= DD5_DI.17
			#625 panStartUFO030101 <= statusUFO030101started
			#626 panStartUFO030102 <= statusUFO030102started
			#627 panAlarm <= alarm
		END_MACRO
		#628 MACRO 8 bit output module 6()
			#629 panErrorTempSensor <= DD1_AI0_error
			#630 panErrorFT0101 <= DD1_AI1_error
			#631 panErrorFT0102 <= DD1_AI2_error
			#632 panErrorQE0102 <= DD1_AI3_error
			#633 panErrorQE0102 <= DD1_AI4_error
			#634 panAlarmHighTemp <= alarmHighTemperature
			#635 panAlarmLowTemp <= alarmLowTemperature
			#636 panND0502dosingError <= ND0502dosingError
		END_MACRO
		#637 MACRO 8 bit output module 7()
			#638 panND0602dosingError <= ND0602dosingError
			#639 panND0603dosingError <= ND0603dosingError
			#640 panND0803dosingError <= ND0803dosingError
			#641 panND0804dosingError <= ND0804dosingError
			#642 panND080301emptyAlarm <= DD1_DI6
			#643 panND080302emptyAlarm <= DD1_DI7
			#644 panN010501alarm <= N010501alarm
			#645 panN010502alarm <= N010502alarm
		END_MACRO
		#646 MACRO 8 bit output module 8()
			#647 panZDE0225errorToOpen <= ZDE0225errorToOpen
			#648 panZDE0225errorToClose <= ZDE0225errorToClose
			#649 panFPKalarm <= DD7_DI.14
			#650 panFPKnotStarted <= FPKnotStarted
			#651 panErrorFPKsensor <= DD1_AI5_error
			#652 panFPKkshe0401errorToOpen <= FPKkshe0401errorToOpen
			#653 panFPKkshe0401errorToClose <= FPKkshe0401errorToClose
			#654 panUFO030101alarm <= statusUFO030101alarm
		END_MACRO
		#655 MACRO 8 bit output module 9()
			#656 panUFO030102alarm <= statusUFO030102alarm
			#657 panFilterFailToRegen020101 <= filterFailToRegen020101
			#658 panErrorToOpenZD0201 <= errorToOpenZD0201
			#659 panErrorToCloseZD0201 <= errorToCloseZD0201
			#660 panErrorToOpenZD0207 <= errorToOpenZD0207
			#661 panErrorToCloseZD0207 <= errorToCloseZD0207
			#662 panFilterFailToRegen020102 <= filterFailToRegen020102
			#663 panErrorToOpenZD0202 <= errorToOpenZD0202
		END_MACRO
		#664 MACRO 8 bit output module 10()
			#665 panErrorToCloseZD0202 <= errorToCloseZD0202
			#666 panErrorToOpenZD0208 <= errorToOpenZD0208
			#667 panErrorToCloseZD0208 <= errorToCloseZD0208
			#668 panFilterFailToRegen020103 <= filterFailToRegen020103
			#669 panErrorToOpenZD0203 <= errorToOpenZD0203
			#670 panErrorToCloseZD0203 <= errorToCloseZD0203
			#671 panErrorToOpenZD0209 <= errorToOpenZD0209
			#672 panErrorToCloseZD0209 <= errorToCloseZD0209
		END_MACRO
		#673 MACRO 8 bit output module 11()
			#674 panFilterFailToRegen020104 <= filterFailToRegen020104
			#675 panErrorToOpenZD0204 <= errorToOpenZD0204
			#676 panErrorToCloseZD0204 <= errorToCloseZD0204
			#677 panErrorToOpenZD0210 <= errorToOpenZD0210
			#678 panErrorToCloseZD0210 <= errorToCloseZD0210
			#679 panFilterFailToRegen020105 <= filterFailToRegen020105
			#680 panErrorToOpenZD0205 <= errorToOpenZD0205
			#681 panErrorToCloseZD0205 <= errorToCloseZD0205
		END_MACRO
		#682 MACRO 8 bit output module 12()
			#683 panErrorToOpenZD0211 <= errorToOpenZD0211
			#684 panErrorToCloseZD0211 <= errorToCloseZD0211
			#685 panFilterFailToRegen020106 <= filterFailToRegen020106
			#686 panErrorToOpenZD0206 <= errorToOpenZD0206
			#687 panErrorToCloseZD0206 <= errorToCloseZD0206
			#688 panErrorToOpenZD0212 <= errorToOpenZD0212
			#689 panErrorToCloseZD0212 <= errorToCloseZD0212
			#690 panFilterFailToRegen020201 <= filterFailToRegen020201
		END_MACRO
		#691 MACRO 8 bit output module 13()
			#692 panErrorToOpenZD0213 <= errorToOpenZD0213
			#693 panErrorToCloseZD0213 <= errorToCloseZD0213
			#694 panErrorToOpenZD0219 <= errorToOpenZD0219
			#695 panErrorToCloseZD0219 <= errorToCloseZD0219
			#696 panFilterFailToRegen020202 <= filterFailToRegen020202
			#697 panErrorToOpenZD0214 <= errorToOpenZD0214
			#698 panErrorToCloseZD0214 <= errorToCloseZD0214
			#699 panErrorToOpenZD0220 <= errorToOpenZD0220
		END_MACRO
		#700 MACRO 8 bit output module 14()
			#701 panErrorToCloseZD0220 <= errorToCloseZD0220
			#702 panFilterFailToRegen020203 <= filterFailToRegen020203
			#703 panErrorToOpenZD0215 <= errorToOpenZD0215
			#704 panErrorToCloseZD0215 <= errorToCloseZD0215
			#705 panErrorToOpenZD0221 <= errorToOpenZD0221
			#706 panErrorToCloseZD0221 <= errorToCloseZD0221
			#707 panFilterFailToRegen020204 <= filterFailToRegen020204
			#708 panErrorToOpenZD0216 <= errorToOpenZD0216
		END_MACRO
		#709 MACRO 8 bit output module 15()
			#710 panErrorToCloseZD0216 <= errorToCloseZD0216
			#711 panErrorToOpenZD0222 <= errorToOpenZD0222
			#712 panErrorToCloseZD0222 <= errorToCloseZD0222
			#713 panFilterFailToRegen020205 <= filterFailToRegen020205
			#714 panErrorToOpenZD0217 <= errorToOpenZD0217
			#715 panErrorToCloseZD0217 <= errorToCloseZD0217
			#716 panErrorToOpenZD0223 <= errorToOpenZD0223
			#717 panErrorToCloseZD0223 <= errorToCloseZD0223
		END_MACRO
		#718 MACRO 8 bit output module 16()
			#719 panFilterFailToRegen020206 <= filterFailToRegen020206
			#720 panErrorToOpenZD0218 <= errorToOpenZD0218
			#721 panErrorToCloseZD0218 <= errorToCloseZD0218
			#722 panErrorToOpenZD0224 <= errorToOpenZD0224
			#723 panErrorToCloseZD0224 <= errorToCloseZD0224
			#724 panAlarmPLKnetwork <= alarmPLKnetwork
			#725 panAlarmND050201 <= alarmND050201
			#726 panAlarmND050202 <= alarmND050202
		END_MACRO
		#727 MACRO 8 bit output module 17()
			#728 panAlarmND060201 <= alarmND060201
			#729 panAlarmND060202 <= alarmND060202
			#730 panAlarmND060301 <= alarmND060301
			#731 panAlarmND060302 <= alarmND060302
			#732 panAlarmND070301 <= alarmND070301
			#733 panAlarmND070302 <= alarmND070302
			#734 panAlarmND080301 <= alarmND080301
			#735 panAlarmND080302 <= alarmND080302
		END_MACRO
		#736 MACRO 8 bit output module 18()
			#737 panAlarmND0804 <= alarmND0804
			#738 panAlarmOGM0104overload <= alarmOGM0104overload
			#739 panAlarmRCHV0203overload <= alarmRCHV0203overload
			#740 panAlarmN040402 <= alarmN040402
			#741 panAlarmN040401 <= alarmN040401
			#742 panAlarmM0604 <= alarmM0604
			#743 panAlarmM0702 <= alarmM0702
			#744 panAlarmM0802 <= alarmM0802
		END_MACRO
		#745 MACRO 8 bit output module 19()
			#746 panAlarmN020401 <= alarmN020401
			#747 panAlarmN020402 <= alarmN020402
			#748 panAlarmFS020101 <= alarmFS020101
			#749 panAlarmFS020102 <= alarmFS020102
			#750 panAlarmFS020103 <= alarmFS020103
			#751 panAlarmFS020104 <= alarmFS020104
			#752 panAlarmFS020105 <= alarmFS020105
			#753 panAlarmFS020106 <= alarmFS020106
		END_MACRO
		#754 MACRO 8 bit output module 20()
			#755 panAlarmFS020201 <= alarmFS020201
			#756 panAlarmFS020202 <= alarmFS020202
			#757 panAlarmFS020203 <= alarmFS020203
			#758 panAlarmFS020204 <= alarmFS020204
			#759 panAlarmFS020205 <= alarmFS020205
			#760 panAlarmFS020206 <= alarmFS020206
			#761 panAlarmZDE0201power <= alarmZDE0201power
			#762 panAlarmZDE0202power <= alarmZDE0202power
		END_MACRO
		#763 MACRO 8 bit output module 21()
			#764 panAlarmZDE0203power <= alarmZDE0203power
			#765 panAlarmZDE0204power <= alarmZDE0204power
			#766 panAlarmZDE0205power <= alarmZDE0205power
			#767 panAlarmZDE0206power <= alarmZDE0206power
			#768 panAlarmZDE0207power <= alarmZDE0207power
			#769 panAlarmZDE0208power <= alarmZDE0208power
			#770 panAlarmZDE0209power <= alarmZDE0209power
			#771 panAlarmZDE0210power <= alarmZDE0210power
		END_MACRO
		#772 MACRO 8 bit output module 22()
			#773 panAlarmZDE0211power <= alarmZDE0211power
			#774 panAlarmZDE0212power <= alarmZDE0212power
			#775 panAlarmZDE0213power <= alarmZDE0213power
			#776 panAlarmZDE0214power <= alarmZDE0214power
			#777 panAlarmZDE0215power <= alarmZDE0215power
			#778 panAlarmZDE0216power <= alarmZDE0216power
			#779 panAlarmZDE0217power <= alarmZDE0217power
			#780 panAlarmZDE0218power <= alarmZDE0218power
		END_MACRO
		#781 MACRO 8 bit output module 23()
			#782 panAlarmZDE0219power <= alarmZDE0219power
			#783 panAlarmZDE0220power <= alarmZDE0220power
			#784 panAlarmZDE0221power <= alarmZDE0221power
			#785 panAlarmZDE0222power <= alarmZDE0222power
			#786 panAlarmZDE0223power <= alarmZDE0223power
			#787 panAlarmZDE0224power <= alarmZDE0224power
			#788 panAlarmZDE0225power <= alarmZDE0225power
			#789 panAlarmKSHE0401power <= alarmKSHE0401power
		END_MACRO
		#790 MACRO 8 bit output module 24()
			#791 panAlarmKNS <= alarmKNS
			#792 panAlarmPowerSocketFS <= alarmPowerSocketFS
			#793 panAlarmKEMvalvesPower <= alarmKEMvalvesPower
			#794 panAlarmEmergencyPressed <= alarmEmergencyPressed
			#795 panAlarmRKF <= alarmRKF
			#796 panUFO0301noFlowAttention <= UFO0301noFlowAttention
			#797 panM0604attention <= M0604attention
			#798 panM0702attention <= M0702attention
		END_MACRO
		#799 MACRO 8 bit output module 25()
			#800 panM0802attention <= M0802attention
			#801 panStatusKNS <= DD6_DI.8
			#802 panND0502statRegimeP1M <= ND0502statRegimeP1M
			#803 panND0502statRegimeP2M <= ND0502statRegimeP2M
			#804 panND0502statRegimeByC <= ND0502statRegimeByC
			#805 panND0502statRegimeByWT <= ND0502statRegimeByWT
			#806 panND0602statRegimeP1M <= ND0602statRegimeP1M
			#807 panND0602statRegimeP2M <= ND0602statRegimeP2M
		END_MACRO
		#808 MACRO 8 bit output module 26()
			#809 panND0602statRegimeByC <= ND0602statRegimeByC
			#810 panND0602statRegimeByWT <= ND0602statRegimeByWT
			#811 panND0603statRegimeP1M <= ND0603statRegimeP1M
			#812 panND0603statRegimeP2M <= ND0603statRegimeP2M
			#813 panND0603statRegimeByC <= ND0603statRegimeByC
			#814 panND0603statRegimeByWT <= ND0603statRegimeByWT
			#815 panND0703statRegimeP1M <= ND0703statRegimeP1M
			#816 panND0703statRegimeP2M <= ND0703statRegimeP2M
		END_MACRO
		#817 MACRO 8 bit output module 27()
			#818 panND0703statRegimeByC <= ND0703statRegimeByC
			#819 panND0703statRegimeByWT <= ND0703statRegimeByWT
			#820 panND0803statRegimeP1M <= ND0803statRegimeP1M
			#821 panND0803statRegimeP2M <= ND0803statRegimeP2M
			#822 panND0803statRegimeByC <= ND0803statRegimeByC
			#823 panND0803statRegimeByWT <= ND0803statRegimeByWT
			#824 panN0105statRegimeP1M <= N0105statRegimeP1M
			#825 panN0105statRegimeP2M <= N0105statRegimeP2M
		END_MACRO
		#826 MACRO 8 bit output module 28()
			#827 panN0105statRegimeByC <= N0105statRegimeByC
			#828 panN0105statRegimeByWT <= N0105statRegimeByWT
			#829 panN0204statRegimeP1M <= N0204statRegimeP1M
			#830 panN0204statRegimeP2M <= N0204statRegimeP2M
			#831 panN0204statRegimeByC <= N0204statRegimeByC
			#832 panN0204statRegimeWT <= N0204statRegimeWT
			#833 panN0404statRegimeP1M <= N0404statRegimeP1M
			#834 panN0404statRegimeP2M <= N0404statRegimeP2M
		END_MACRO
		#835 MACRO 8 bit output module 29()
			#836 panN0404statRegimeByC <= N0404statRegimeByC
			#837 panN0404statRegimeWT <= N0404statRegimeWT
			#838 panUFO0301statRegimeP1M <= UFO0301statRegimeP1M
			#839 panUFO0301statRegimeP2M <= UFO0301statRegimeP2M
			#840 panUFO0301statRegimeByC <= UFO0301statRegimeByC
			#841 panUFO0301statRegimeWT <= UFO0301statRegimeWT
			#842 panZDE0225open <= DD9_DI.0
			#843 panZDE0201open <= DD7_DI.16
		END_MACRO
		#844 MACRO 8 bit output module 30()
			#845 panZDE0201close <= DD7_DI.17
			#846 panZDE0202open <= DD7_DI.18
			#847 panZDE0202close <= DD7_DI.19
			#848 panZDE0203open <= DD7_DI.20
			#849 panZDE0203close <= DD7_DI.21
			#850 panZDE0204open <= DD7_DI.22
			#851 panZDE0204close <= DD7_DI.23
			#852 panZDE0205open <= DD7_DI.24
		END_MACRO
		#853 MACRO 8 bit output module 31()
			#854 panZDE0205close <= DD7_DI.25
			#855 panZDE0206open <= DD7_DI.26
			#856 panZDE0206close <= DD7_DI.27
			#857 panZDE0207open <= DD7_DI.28
			#858 panZDE0207close <= DD7_DI.29
			#859 panZDE0208open <= DD7_DI.30
			#860 panZDE0208close <= DD7_DI.31
			#861 panZDE0209open <= DD8_DI.0
		END_MACRO
		#862 MACRO 8 bit output module 32()
			#863 panZDE0209close <= DD8_DI.1
			#864 panZDE0210open <= DD8_DI.2
			#865 panZDE0210close <= DD8_DI.3
			#866 panZDE0211open <= DD8_DI.4
			#867 panZDE0211close <= DD8_DI.5
			#868 panZDE0212open <= DD8_DI.6
			#869 panZDE0212close <= DD8_DI.7
			#870 panZDE0213open <= DD8_DI.8
		END_MACRO
		#871 MACRO 8 bit output module 33()
			#872 panZDE0213close <= DD8_DI.9
			#873 panZDE0214open <= DD8_DI.10
			#874 panZDE0214close <= DD8_DI.11
			#875 panZDE0215open <= DD8_DI.12
			#876 panZDE0215close <= DD8_DI.13
			#877 panZDE0216open <= DD8_DI.14
			#878 panZDE0216close <= DD8_DI.15
			#879 panZDE0217open <= DD8_DI.16
		END_MACRO
		#880 MACRO 8 bit output module 34()
			#881 panZDE0217close <= DD8_DI.17
			#882 panZDE0218open <= DD8_DI.18
			#883 panZDE0218close <= DD8_DI.19
			#884 panZDE0219open <= DD8_DI.20
			#885 panZDE0219close <= DD8_DI.21
			#886 panZDE0220open <= DD8_DI.22
			#887 panZDE0220close <= DD8_DI.23
			#888 panZDE0221open <= DD8_DI.24
		END_MACRO
		#889 MACRO 8 bit output module 35()
			#890 panZDE0221close <= DD8_DI.25
			#891 panZDE0222open <= DD8_DI.26
			#892 panZDE0222close <= DD8_DI.27
			#893 panZDE0223open <= DD8_DI.28
			#894 panZDE0223close <= DD8_DI.29
			#895 panZDE0224open <= DD8_DI.30
			#896 panZDE0224close <= DD8_DI.31
			#897 panZDE0225close <= DD9_DI.1
		END_MACRO
		#898 MACRO 8 bit output module 36x()
			#899 panKSHE0401close <= DD9_DI.3
			#900 panZDE0301open <= DD1_DI12
			#901 panZDE0301close <= DD1_DI13
			#902 panZDE0302open <= DD1_DI14
			#903 panZDE0302close <= DD1_DI15
			#904 panErrorToOpenZDE0301 <= errorToOpenZDE0301
			#905 panErrorToCloseZDE0301 <= errorToCloseZDE0301
			#906 panErrorToOpenZDE0302 <= errorToOpenZDE0302
		END_MACRO
		#907 panErrorToCloseZDE0302 <= errorToCloseZDE0302
		#908 panAlarmZDE0301power <= alarmZDE0301power
		#909 panAlarmZDE0302power <= alarmZDE0302power
		#910 panUFO030101danger <= statusUFO030101danger
		#911 panUFO030102danger <= statusUFO030102danger
		#912 panUFO030101distantMode <= statusUFO030101distantMode
		#913 panUFO030102distantMode <= statusUFO030102distantMode
	END_MACRO
	#914 MACRO PFW регистры на чтение из панели (управление ПЛК)()
		#915 MUL(panTimeToOpenCloseValve, 1000)
		#916 REAL_TO_TIME(#915)
		#917 TimeToOpenCloseValve <= #916
		#918 maxTemperature <= panMaxTemperature
		#919 minTemperature <= panMinTemperature
		#920 ND0502setMaxDosVal <= panND0502setMaxDosVal
		#921 ND0502setKoefProp <= panND0502setKoefProp
		#922 ND0602setMaxDosVal <= panND0602setMaxDosVal
		#923 ND0602setKoefProp <= panND0602setKoefProp
		#924 ND0603setMaxDosVal <= panND0603setMaxDosVal
		#925 ND0603setKoefProp <= panND0603setKoefProp
		#926 ND0703pHsetValue <= panND0703pHsetValue
		#927 ND0703YoutManual <= panND0703YoutManual
		#928 ND0703koeffI <= panND0703koeffI
		#929 ND0703koeffD <= panND0703koeffD
		#930 ND0703koeffP <= panND0703koeffP
		#931 ND0803setMaxDosVal <= panND0803setMaxDosVal
		#932 ND0803setKoefProp <= panND0803setKoefProp
		#933 ND0804doseValue <= panND0804doseValue
		#934 N0105flowSetValue <= panN0105flowSetValue
		#935 N0105YoutManual <= panN0105YoutManual
		#936 N0105koeffI <= panN0105koeffI
		#937 N0105koeffD <= panN0105koeffD
		#938 N0105koeffP <= panN0105koeffP
		#939 FQS0301impulsValue <= panFQS0301impulsValue
		#940 FQS0301correction <= panFQS0301correction
		#941 MUL(panFPKtimeToWork, 1000)
		#942 REAL_TO_TIME(#941)
		#943 FPKtimeToWork <= #942
		#944 MUL(panFPKnotStartedTime, 1000)
		#945 REAL_TO_TIME(#944)
		#946 FPKnotStartedTime <= #945
		#947 FPKmaxPressureValue <= panFPKmaxPressureValue
		#948 filterValueToRegen <= panFilterValueToRegen
	END_MACRO
	#949 MACRO PSB регистры на чтение из панели (управление ПЛК)()
		(* PSB регистры на чтение из панели (управление ПЛК) *)
		#950 MACRO 8 bit input module 1()
			#1280 alarmReset <= panAlarmResetButton
			#1281 ND0502resetCountP1 <= panND0502resetCountP1
			#1282 ND0502resetCountP2 <= panND0502resetCountP2
			#1283 ND0502resetWorkTimeP1 <= panND0502resetWorkTimeP1
			#1284 ND0502resetWorkTimeP2 <= panND0502resetWorkTimeP2
			#1285 ND0502regimeP1M <= panND0502regimeP1M
			#1286 ND0502regimeP2M <= panND0502regimeP2M
			#1287 ND0502regimeByC <= panND0502regimeByC
		END_MACRO
		#951 MACRO 8 bit input module 2()
			#1288 ND0502regimeByWT <= panND0502regimeByWT
			#1289 ND0602resetCountP1 <= panND0602resetCountP1
			#1290 ND0602resetCountP2 <= panND0602resetCountP2
			#1291 ND0602resetWorkTimeP1 <= panND0602resetWorkTimeP1
			#1292 ND0602resetWorkTimeP2 <= panND0602resetWorkTimeP2
			#1293 ND0602regimeP1M <= panND0602regimeP1M
			#1294 ND0602regimeP2M <= panND0602regimeP2M
			#1295 ND0602regimeByC <= panND0602regimeByC
		END_MACRO
		#952 MACRO 8 bit input module 3()
			#1296 ND0602regimeByWT <= panND0602regimeByWT
			#1297 ND0603resetCountP1 <= panND0603resetCountP1
			#1298 ND0603resetCountP2 <= panND0603resetCountP2
			#1299 ND0603resetWorkTimeP1 <= panND0603resetWorkTimeP1
			#1300 ND0603resetWorkTimeP2 <= panND0603resetWorkTimeP2
			#1301 ND0603regimeP1M <= panND0603regimeP1M
			#1302 ND0603regimeP2M <= panND0603regimeP2M
			#1303 ND0603regimeByC <= panND0603regimeByC
		END_MACRO
		#953 MACRO 8 bit input module 4()
			#1304 ND0603regimeByWT <= panND0603regimeByWT
			#1305 ND0703resetCountP1 <= panND0703resetCountP1
			#1306 ND0703resetCountP2 <= panND0703resetCountP2
			#1307 ND0703resetWorkTimeP1 <= panND0703resetWorkTimeP1
			#1308 ND0703resetWorkTimeP2 <= panND0703resetWorkTimeP2
			#1309 ND0703regimeP1M <= panND0703regimeP1M
			#1310 ND0703regimeP2M <= panND0703regimeP2M
			#1311 ND0703regimeByC <= panND0703regimeByC
		END_MACRO
		#954 MACRO 8 bit input module 5()
			#1312 ND0703regimeByWT <= panND0703regimeByWT
			#1313 ND0703YmanAuto <= panND0703YmanAuto
			#1314 ND0803resetCountP1 <= panND0803resetCountP1
			#1315 ND0803resetCountP2 <= panND0803resetCountP2
			#1316 ND0803resetWorkTimeP1 <= panND0803resetWorkTimeP1
			#1317 ND0803resetWorkTimeP2 <= panND0803resetWorkTimeP2
			#1318 ND0803regimeP1M <= panND0803regimeP1M
			#1319 ND0803regimeP2M <= panND0803regimeP2M
		END_MACRO
		#955 MACRO 8 bit input module 6()
			#1320 ND0803regimeByC <= panND0803regimeByC
			#1321 ND0803regimeByWT <= panND0803regimeByWT
			#1322 N0105resetCountP1 <= panN0105resetCountP1
			#1323 N0105resetCountP2 <= panN0105resetCountP2
			#1324 N0105resetWorkTimeP1 <= panN0105resetWorkTimeP1
			#1325 N0105resetWorkTimeP2 <= panN0105resetWorkTimeP2
			#1326 N0105regimeByC <= panN0105regimeByC
			#1327 N0105regimeByWT <= panN0105regimeByWT
		END_MACRO
		#956 MACRO 8 bit input module 7()
			#1328 N0105YmanAuto <= panN0105YmanAuto
			#1329 N0204resetCountP1 <= panN0204resetCountP1
			#1330 N0204resetCountP2 <= panN0204resetCountP2
			#1331 N0204resetWorkTimeP1 <= panN0204resetWorkTimeP1
			#1332 N0204resetWorkTimeP2 <= panN0204resetWorkTimeP2
			#1333 N0204regimeP1M <= panN0204regimeP1M
			#1334 N0204regimeP2M <= panN0204regimeP2M
			#1335 N0204regimeByC <= panN0204regimeByC
		END_MACRO
		#957 MACRO 8 bit input module 8()
			#1336 N0204regimeWT <= panN0204regimeWT
			#1337 UFO0301resetCountP1 <= panUFO0301resetCountP1
			#1338 UFO0301resetCountP2 <= panUFO0301resetCountP2
			#1339 UFO0301resetWorkTimeP1 <= panUFO0301resetWorkTimeP1
			#1340 UFO0301resetWorkTimeP2 <= panUFO0301resetWorkTimeP2
			#1341 UFO0301regimeP1M <= panUFO0301regimeP1M
			#1342 UFO0301regimeP2M <= panUFO0301regimeP2M
			#1343 UFO0301regimeByC <= panUFO0301regimeByC
		END_MACRO
		#958 MACRO 8 bit input module 9()
			#1344 UFO0301regimeWT <= panUFO0301regimeWT
			#1345 N0404resetCountP1 <= panN0404resetCountP1
			#1346 N0404resetCountP2 <= panN0404resetCountP2
			#1347 N0404resetWorkTimeP1 <= panN0404resetWorkTimeP1
			#1348 N0404resetWorkTimeP2 <= panN0404resetWorkTimeP2
			#1349 N0404regimeP1M <= panN0404regimeP1M
			#1350 N0404regimeP2M <= panN0404regimeP2M
			#1351 N0404regimeByC <= panN0404regimeByC
		END_MACRO
		#959 MACRO 8 bit input module 10-11()
			(* одули 10 и 11 заполнены переменными для тестирования задвижек. / Здесь они не показаны, т.к. спешка. / Они вставлены напрямую в макросы управления промывкой фильтров. / testValvesFS020101 - testValvesFS020206 (PSB612-623) *)
			#1352 N0404regimeWT <= panN0404regimeWT
			#1353 FQS0301reset <= panFQS0301reset
			#1354 FQS0301addCorrection <= panFQS0301addCorrection
			#1355 FQS0301deleteCorrection <= panFQS0301deleteCorrection
		END_MACRO
		#960 testKSHE0401 <= panTestKSHE0401
		#961 testZDE0225 <= panTestZDE0225
		#962 testZDE03 <= panTestZDE03
		#963 manualZDE0301 <= panManualZDE0301
		#964 manualZDE0302 <= panManualZDE0302
	END_MACRO
END_MACRO
#965 NOT(DD6_DI.13)
#966 alarmRCHV0203overload <= #965
#967 NOT(DD9_DI.5)
#968 alarmZDE0202power <= #967
#969 NOT(DD9_DI.26)
#970 alarmZDE0223power <= #969
#971 MACRO переменные на диспетчеризацию()
	#972 remFT0101value <= DD1_AI1_FT0101value
	#973 remFQS0301totalAmount <= FQS0301totalAmount
	#974 remTemperatureValue <= temperatureValue
	#975 remStatusN010501started <= N0105statStartedP1
	#976 remStatusN010502started <= N0105statStartedP2
	#977 remStatusUFO030101started <= statusUFO030101started
	#978 remStatusUFO030102started <= statusUFO030102started
	#979 remAlarm <= Alarm
	#980 remN010501alarm <= N010501alarm
	#981 remN010502alarm <= N010502alarm
	#982 remFPKalarm <= DD7_DI.14
	#983 remUFO030101alarm <= statusUFO030101alarm
	#984 remUFO030102alarm <= statusUFO030102alarm
	#985 remAlarmEmergencyPressed <= alarmEmergencyPressed
	#986 remAlarmOOGM0104overload <= DD6_DI.11
	#987 remAlarmRCHV0203overload <= DD6_DI.13
END_MACRO
#988 NOT(DD5_DI.14)
#989 alarmN040402 <= #988
#990 NOT(DD9_DI.6)
#991 alarmZDE0203power <= #990
#992 NOT(DD9_DI.27)
#993 alarmZDE0224power <= #992
#994 NOT(DD5_DI.15)
#995 alarmN040401 <= #994
#996 NOT(DD9_DI.7)
#997 alarmZDE0204power <= #996
#998 NOT(DD9_DI.28)
#999 alarmZDE0225power <= #998
#1000 NOT(DD5_DI.20)
#1001 alarmM0604 <= #1000
#1002 NOT(DD9_DI.8)
#1003 alarmZDE0205power <= #1002
#1004 NOT(DD9_DI.29)
#1005 alarmKSHE0401power <= #1004
#1006 NOT(DD5_DI.22)
#1007 alarmM0702 <= #1006
#1008 NOT(DD9_DI.9)
#1009 alarmZDE0206power <= #1008
#1010 NOT(DD6_DI.9)
#1011 alarmKNS <= #1010
#1012 NOT(DD5_DI.24)
#1013 alarmM0802 <= #1012
#1014 NOT(DD9_DI.10)
#1015 alarmZDE0207power <= #1014
#1016 NOT(DD6_DI.17)
#1017 alarmPowerSocketFS <= #1016
#1018 NOT(DD5_DI.7)
#1019 alarmN020401 <= #1018
#1020 NOT(DD9_DI.11)
#1021 alarmZDE0208power <= #1020
#1022 NOT(DD6_DI.18)
#1023 alarmKEMvalvesPower <= #1022
#1024 NOT(DD5_DI.8)
#1025 alarmN020402 <= #1024
#1026 NOT(DD9_DI.12)
#1027 alarmZDE0209power <= #1026
#1028 NOT(DD1_DI4)
#1029 alarmEmergencyPressed <= #1028
#1030 GT(DD1_AI2_FT0102value, 0)
#1031 filterPulserGen:PulsePerSec(start: #1030)
#1032 DIV(DD1_AI2_FT0102value, 3600)
#1033 ADD(EN: #1031.out, #1032, filterTotalAmountFT0102)
#1034 filterTotalAmountFT0102 <= #1033
#1035 NOT(DD6_DI.21)
#1036 alarmFS020101 <= #1035
#1037 NOT(DD9_DI.13)
#1038 alarmZDE0210power <= #1037
#1039 NOT(DD1_DI5)
#1040 alarmRKF <= #1039
#1041 NOT(DD9_DI.30)
#1042 alarmZDE0301power <= #1041
#1043 NOT(DD9_DI.31)
#1044 alarmZDE0302power <= #1043
#1045 MOVE(EN: filterTotalAmountReset, 0)
#1046 filterTotalAmountFT0102 <= #1045
#1047 SUB(filterValueToRegen, filterTotalAmountFT0102)
#1048 volumeToRegen <= #1047
#1049 GE(filterTotalAmountFT0102, filterValueToRegen)
#1050 MACRO управление промывкой фильтра ФС02.01.01(pin 1 "сигнал на промывку": #1049, pin 2 "авария фильтра": DD6_DI.21, pin 3 "подтверждение промывки": DD6_DI.20, pin 4 "сброс аварий": alarmReset, pin 5 "начать очередь снова": filterStartNewQueue, pin 6 "ЗДЭ02.01 открыта": DD7_DI.16, pin 7 "ЗДЭ02.01 закрыта": DD7_DI.17, pin 8 "ЗДЭ02.07 открыта": DD7_DI.28, pin 9 "ЗДЭ02.07 закрыта": DD7_DI.29, pin 10 "время движения ЗДЭ": timeToOpenCloseValve, pin 11 "авария питания ЗДЭ02.01": DD9_DI.4, pin 12 "авария питания ЗДЭ02.07": DD9_DI.10)
	(* <- выход использовать в / последнем фильтре для / начала очереди заново *)
	(* если открыт = промывка *)
	(* если открыт = фильтрация *)
	out 1 "следующий в очереди" <= #1053.output
	out 2 "промыть ФС02.01.01" <= #1052
	#1051 ZD0201:SimpleValve(inputOpen: NOT #1052, inputClose: #1052, statusOpen: pin 6, statusClose: pin 7, reset: pin 4, timeToOpenClose: pin 10)
	out 6 "открыть ЗДЭ02.01" <= #1051.outputOpen
	out 7 "закрыть ЗДЭ02.01" <= #1051.outputClose
	out 8 "авария открытия ЗДЭ02.01" <= #1051.errorToOpen
	#1052 OR(panTestValvesFS020101, #1053.regenFilterOUT)
	out 9 "авария закрытия ЗДЭ02.01" <= #1051.errorToClose
	#1053 FS020101manager:FilterQueueManager(input: pin 1, filterAlarm: #1054, regenFilterStatus: pin 3, alarmReset: pin 4, startNextLoop: pin 5)
	#1054 OR(alarmZD020107, pin 2, pin 11, pin 12)
	out 3 "ФС02.01.01 промыт" <= #1053.regenerated
	out 4 "не удалось промыть" <= #1053.failToRegen
	#1055 OR(#1051.errorToOpen, #1051.errorToClose, #1057.errorToOpen, #1057.errorToClose)
	#1056 alarmZD020107 <= #1055
	out 5 "сброс счетчика" <= #1053.counterReset
	#1057 ZD0207:SimpleValve(inputOpen: #1052, inputClose: NOT #1052, statusOpen: pin 8, statusClose: pin 9, reset: pin 4, timeToOpenClose: pin 10)
	out 10 "открыть ЗДЭ02.07" <= #1057.outputOpen
	out 11 "закрыть ЗДЭ02.07" <= #1057.outputClose
	out 12 "авария открытия ЗДЭ02.07" <= #1057.errorToOpen
	out 13 "авария закрытия ЗДЭ02.07" <= #1057.errorToClose
END_MACRO
#1058 DD2_DO.4 <= #1050.out 2
#1059 regeneratedFS020101 <= #1050.out 3
#1060 filterFailToRegen020101 <= #1050.out 4
#1061 filterTotalAmountReset <= #1050.out 5
#1062 DD2_DO.16 <= #1050.out 6
#1063 DD2_DO.17 <= #1050.out 7
#1064 errorToOpenZD0201 <= #1050.out 8
#1065 errorToCloseZD0201 <= #1050.out 9
#1066 DD2_DO.28 <= #1050.out 10
#1067 DD2_DO.29 <= #1050.out 11
#1068 errorToOpenZD0207 <= #1050.out 12
#1069 errorToCloseZD0207 <= #1050.out 13
#1070 MACRO управление промывкой фильтра ФС02.01.02(pin 1 "сигнал на промывку": #1050.out 1, pin 2 "авария фильтра": DD6_DI.23, pin 3 "подтверждение промывки": DD6_DI.22, pin 4 "сброс аварий": alarmReset, pin 5 "начать очередь снова": filterStartNewQueue, pin 6 "ЗДЭ02.02 открыта": DD7_DI.18, pin 7 "ЗДЭ02.02 закрыта": DD7_DI.19, pin 8 "ЗДЭ02.08 открыта": DD7_DI.30, pin 9 "ЗДЭ02.08 закрыта": DD7_DI.31, pin 10 "время движения ЗДЭ": timeToOpenCloseValve, pin 11 "авария питания ЗДЭ02.02": DD9_DI.5, pin 12 "авария питания ЗДЭ02.08": DD9_DI.11)
	(* <- выход использовать в / последнем фильтре для / начала очереди заново *)
	(* если открыт = промывка *)
	(* если открыт = фильтрация *)
	out 1 "следующий в очереди" <= #1073.output
	out 2 "промыть ФС02.01.02" <= #1072
	#1071 ZD0202:SimpleValve(inputOpen: NOT #1072, inputClose: #1072, statusOpen: pin 6, statusClose: pin 7, reset: pin 4, timeToOpenClose: pin 10)
	out 5 "открыть ЗДЭ02.02" <= #1071.outputOpen
	out 6 "закрыть ЗДЭ02.02" <= #1071.outputClose
	out 7 "авария открытия ЗДЭ02.02" <= #1071.errorToOpen
	#1072 OR(panTestValvesFS020102, #1073.regenFilterOUT)
	out 8 "авария закрытия ЗДЭ02.02" <= #1071.errorToClose
	#1073 FS020102manager:FilterQueueManager(input: pin 1, filterAlarm: #1074, regenFilterStatus: pin 3, alarmReset: pin 4, startNextLoop: pin 5)
	#1074 OR(alarmZD020208, pin 2, pin 11, pin 12)
	#1075 OR(#1071.errorToOpen, #1071.errorToClose, #1077.errorToOpen, #1077.errorToClose)
	#1076 alarmZD020208 <= #1075
	out 3 "ФС02.01.02 промыт" <= #1073.regenerated
	out 4 "не удалось промыть" <= #1073.failToRegen
	#1077 ZD0208:SimpleValve(inputOpen: #1072, inputClose: NOT #1072, statusOpen: pin 8, statusClose: pin 9, reset: pin 4, timeToOpenClose: pin 10)
	out 9 "открыть ЗДЭ02.08" <= #1077.outputOpen
	out 10 "закрыть ЗДЭ02.08" <= #1077.outputClose
	out 11 "авария открытия ЗДЭ02.08" <= #1077.errorToOpen
	out 12 "авария закрытия ЗДЭ02.08" <= #1077.errorToClose
END_MACRO
#1078 DD2_DO.5 <= #1070.out 2
#1079 regeneratedFS020102 <= #1070.out 3
#1080 filterFailToRegen020102 <= #1070.out 4
#1081 DD2_DO.18 <= #1070.out 5
#1082 DD2_DO.19 <= #1070.out 6
#1083 errorToOpenZD0202 <= #1070.out 7
#1084 errorToCloseZD0202 <= #1070.out 8
#1085 DD2_DO.30 <= #1070.out 9
#1086 DD2_DO.31 <= #1070.out 10
#1087 errorToOpenZD0208 <= #1070.out 11
#1088 errorToCloseZD0208 <= #1070.out 12
#1089 MACRO управление промывкой фильтра ФС02.01.03(pin 1 "сигнал на промывку": #1070.out 1, pin 2 "авария фильтра": DD6_DI.25, pin 3 "подтверждение промывки": DD6_DI.24, pin 4 "сброс аварий": alarmReset, pin 5 "начать очередь снова": filterStartNewQueue, pin 6 "ЗДЭ02.03 открыта": DD7_DI.20, pin 7 "ЗДЭ02.03 закрыта": DD7_DI.21, pin 8 "ЗДЭ02.09 открыта": DD8_DI.0, pin 9 "ЗДЭ02.09 закрыта": DD8_DI.1, pin 10 "время движения ЗДЭ": timeToOpenCloseValve, pin 11 "авария питания ЗДЭ02.03": DD9_DI.6, pin 12 "авария питания ЗДЭ02.09": DD9_DI.12)
	(* <- выход использовать в / последнем фильтре для / начала очереди заново *)
	(* если открыт = промывка *)
	(* если открыт = фильтрация *)
	out 1 "следующий в очереди" <= #1092.output
	out 2 "промыть ФС02.01.03" <= #1091
	#1090 ZD0203:SimpleValve(inputOpen: NOT #1091, inputClose: #1091, statusOpen: pin 6, statusClose: pin 7, reset: pin 4, timeToOpenClose: pin 10)
	out 5 "открыть ЗДЭ02.03" <= #1090.outputOpen
	out 6 "закрыть ЗДЭ02.03" <= #1090.outputClose
	out 7 "авария открытия ЗДЭ02.03" <= #1090.errorToOpen
	#1091 OR(panTestValvesFS020103, #1092.regenFilterOUT)
	out 8 "авария закрытия ЗДЭ02.03" <= #1090.errorToClose
	#1092 FS020103manager:FilterQueueManager(input: pin 1, filterAlarm: #1093, regenFilterStatus: pin 3, alarmReset: pin 4, startNextLoop: pin 5)
	#1093 OR(alarmZD020309, pin 2, pin 11, pin 12)
	#1094 OR(#1090.errorToOpen, #1090.errorToClose, #1096.errorToOpen, #1096.errorToClose)
	#1095 alarmZD020309 <= #1094
	out 3 "ФС02.01.03 промыт" <= #1092.regenerated
	out 4 "не удалось промыть" <= #1092.failToRegen
	#1096 ZD0209:SimpleValve(inputOpen: #1091, inputClose: NOT #1091, statusOpen: pin 8, statusClose: pin 9, reset: pin 4, timeToOpenClose: pin 10)
	out 9 "открыть ЗДЭ02.09" <= #1096.outputOpen
	out 10 "закрыть ЗДЭ02.09" <= #1096.outputClose
	out 11 "авария открытия ЗДЭ02.09" <= #1096.errorToOpen
	out 12 "авария закрытия ЗДЭ02.09" <= #1096.errorToClose
END_MACRO
#1097 DD2_DO.6 <= #1089.out 2
#1098 regeneratedFS020103 <= #1089.out 3
#1099 filterFailToRegen020103 <= #1089.out 4
#1100 DD2_DO.20 <= #1089.out 5
#1101 DD2_DO.21 <= #1089.out 6
#1102 errorToOpenZD0203 <= #1089.out 7
#1103 errorToCloseZD0203 <= #1089.out 8
#1104 DD3_DO.0 <= #1089.out 9
#1105 DD3_DO.1 <= #1089.out 10
#1106 errorToOpenZD0209 <= #1089.out 11
#1107 errorToCloseZD0209 <= #1089.out 12
#1108 MACRO управление промывкой фильтра ФС02.01.04(pin 1 "сигнал на промывку": #1089.out 1, pin 2 "авария фильтра": DD6_DI.27, pin 3 "подтверждение промывки": DD6_DI.26, pin 4 "сброс аварий": alarmReset, pin 5 "начать очередь снова": filterStartNewQueue, pin 6 "ЗДЭ02.04 открыта": DD7_DI.22, pin 7 "ЗДЭ02.04 закрыта": DD7_DI.23, pin 8 "ЗДЭ02.10 открыта": DD8_DI.2, pin 9 "ЗДЭ02.10 закрыта": DD8_DI.3, pin 10 "время движения ЗДЭ": timeToOpenCloseValve, pin 11 "авария питания ЗДЭ02.04": DD9_DI.7, pin 12 "авария питания ЗДЭ02.10": DD9_DI.13)
	(* <- выход использовать в / последнем фильтре для / начала очереди заново *)
	(* если открыт = промывка *)
	(* если открыт = фильтрация *)
	out 1 "следующий в очереди" <= #1111.output
	out 2 "промыть ФС02.01.04" <= #1110
	#1109 ZD0204:SimpleValve(inputOpen: NOT #1110, inputClose: #1110, statusOpen: pin 6, statusClose: pin 7, reset: pin 4, timeToOpenClose: pin 10)
	out 5 "открыть ЗДЭ02.04" <= #1109.outputOpen
	out 6 "закрыть ЗДЭ02.04" <= #1109.outputClose
	out 7 "авария открытия ЗДЭ02.04" <= #1109.errorToOpen
	#1110 OR(panTestValvesFS020104, #1111.regenFilterOUT)
	out 8 "авария закрытия ЗДЭ02.04" <= #1109.errorToClose
	#1111 FS020104manager:FilterQueueManager(input: pin 1, filterAlarm: #1112, regenFilterStatus: pin 3, alarmReset: pin 4, startNextLoop: pin 5)
	#1112 OR(alarmZD020410, pin 2, pin 11, pin 12)
	#1113 OR(#1109.errorToOpen, #1109.errorToClose, #1115.errorToOpen, #1115.errorToClose)
	#1114 alarmZD020410 <= #1113
	out 3 "ФС02.01.04 промыт" <= #1111.regenerated
	out 4 "не удалось промыть" <= #1111.failToRegen
	#1115 ZD0210:SimpleValve(inputOpen: #1110, inputClose: NOT #1110, statusOpen: pin 8, statusClose: pin 9, reset: pin 4, timeToOpenClose: pin 10)
	out 9 "открыть ЗДЭ02.10" <= #1115.outputOpen
	out 10 "закрыть ЗДЭ02.10" <= #1115.outputClose
	out 11 "авария открытия ЗДЭ02.10" <= #1115.errorToOpen
	out 12 "авария закрытия ЗДЭ02.10" <= #1115.errorToClose
END_MACRO
#1116 DD2_DO.7 <= #1108.out 2
#1117 regeneratedFS020104 <= #1108.out 3
#1118 filterFailToRegen020104 <= #1108.out 4
#1119 DD2_DO.22 <= #1108.out 5
#1120 DD2_DO.23 <= #1108.out 6
#1121 errorToOpenZD0204 <= #1108.out 7
#1122 errorToCloseZD0204 <= #1108.out 8
#1123 DD3_DO.2 <= #1108.out 9
#1124 DD3_DO.3 <= #1108.out 10
#1125 errorToOpenZD0210 <= #1108.out 11
#1126 errorToCloseZD0210 <= #1108.out 12
#1127 MACRO управление промывкой фильтра ФС02.01.05(pin 1 "сигнал на промывку": #1108.out 1, pin 2 "авария фильтра": DD6_DI.29, pin 3 "подтверждение промывки": DD6_DI.28, pin 4 "сброс аварий": alarmReset, pin 5 "начать очередь снова": filterStartNewQueue, pin 6 "ЗДЭ02.05 открыта": DD7_DI.24, pin 7 "ЗДЭ02.05 закрыта": DD7_DI.25, pin 8 "ЗДЭ02.11 открыта": DD8_DI.4, pin 9 "ЗДЭ02.11 закрыта": DD8_DI.5, pin 10 "время движения ЗДЭ": timeToOpenCloseValve, pin 11 "авария питания ЗДЭ02.05": DD9_DI.8, pin 12 "авария питания ЗДЭ02.11": DD9_DI.14)
	(* <- выход использовать в / последнем фильтре для / начала очереди заново *)
	(* если открыт = промывка *)
	(* если открыт = фильтрация *)
	out 1 "следующий в очереди" <= #1130.output
	out 2 "промыть ФС02.01.05" <= #1129
	#1128 ZD0205:SimpleValve(inputOpen: NOT #1129, inputClose: #1129, statusOpen: pin 6, statusClose: pin 7, reset: pin 4, timeToOpenClose: pin 10)
	out 5 "открыть ЗДЭ02.05" <= #1128.outputOpen
	out 6 "закрыть ЗДЭ02.05" <= #1128.outputClose
	out 7 "авария открытия ЗДЭ02.05" <= #1128.errorToOpen
	#1129 OR(panTestValvesFS020105, #1130.regenFilterOUT)
	out 8 "авария закрытия ЗДЭ02.05" <= #1128.errorToClose
	#1130 FS020105manager:FilterQueueManager(input: pin 1, filterAlarm: #1131, regenFilterStatus: pin 3, alarmReset: pin 4, startNextLoop: pin 5)
	#1131 OR(alarmZD020511, pin 2, pin 11, pin 12)
	#1132 OR(#1128.errorToOpen, #1128.errorToClose, #1134.errorToOpen, #1134.errorToClose)
	#1133 alarmZD020511 <= #1132
	out 3 "ФС02.01.05 промыт" <= #1130.regenerated
	out 4 "не удалось промыть" <= #1130.failToRegen
	#1134 ZD0211:SimpleValve(inputOpen: #1129, inputClose: NOT #1129, statusOpen: pin 8, statusClose: pin 9, reset: pin 4, timeToOpenClose: pin 10)
	out 9 "открыть ЗДЭ02.11" <= #1134.outputOpen
	out 10 "закрыть ЗДЭ02.11" <= #1134.outputClose
	out 11 "авария открытия ЗДЭ02.11" <= #1134.errorToOpen
	out 12 "авария закрытия ЗДЭ02.11" <= #1134.errorToClose
END_MACRO
#1135 DD2_DO.8 <= #1127.out 2
#1136 regeneratedFS020105 <= #1127.out 3
#1137 filterFailToRegen020105 <= #1127.out 4
#1138 DD2_DO.24 <= #1127.out 5
#1139 DD2_DO.25 <= #1127.out 6
#1140 errorToOpenZD0205 <= #1127.out 7
#1141 errorToCloseZD0205 <= #1127.out 8
#1142 DD3_DO.4 <= #1127.out 9
#1143 DD3_DO.5 <= #1127.out 10
#1144 errorToOpenZD0211 <= #1127.out 11
#1145 errorToCloseZD0211 <= #1127.out 12
#1146 MACRO управление промывкой фильтра ФС02.01.06(pin 1 "сигнал на промывку": #1127.out 1, pin 2 "авария фильтра": DD6_DI.31, pin 3 "подтверждение промывки": DD6_DI.30, pin 4 "сброс аварий": alarmReset, pin 5 "начать очередь снова": filterStartNewQueue, pin 6 "ЗДЭ02.06 открыта": DD7_DI.26, pin 7 "ЗДЭ02.06 закрыта": DD7_DI.27, pin 8 "ЗДЭ02.12 открыта": DD8_DI.6, pin 9 "ЗДЭ02.12 закрыта": DD8_DI.7, pin 10 "время движения ЗДЭ": timeToOpenCloseValve, pin 11 "авария питания ЗДЭ02.06": DD9_DI.9, pin 12 "авария питания ЗДЭ02.12": DD9_DI.15)
	(* <- выход использовать в / последнем фильтре для / начала очереди заново *)
	(* если открыт = промывка *)
	(* если открыт = фильтрация *)
	out 1 "следующий в очереди" <= #1149.output
	out 2 "промыть ФС02.01.06" <= #1148
	#1147 ZD0206:SimpleValve(inputOpen: NOT #1148, inputClose: #1148, statusOpen: pin 6, statusClose: pin 7, reset: pin 4, timeToOpenClose: pin 10)
	out 5 "открыть ЗДЭ02.06" <= #1147.outputOpen
	out 6 "закрыть ЗДЭ02.06" <= #1147.outputClose
	out 7 "авария открытия ЗДЭ02.06" <= #1147.errorToOpen
	#1148 OR(panTestValvesFS020106, #1149.regenFilterOUT)
	out 8 "авария закрытия ЗДЭ02.06" <= #1147.errorToClose
	#1149 FS020106manager:FilterQueueManager(input: pin 1, filterAlarm: #1150, regenFilterStatus: pin 3, alarmReset: pin 4, startNextLoop: pin 5)
	#1150 OR(alarmZD020612, pin 2, pin 11, pin 12)
	#1151 OR(#1147.errorToOpen, #1147.errorToClose, #1153.errorToOpen, #1153.errorToClose)
	#1152 alarmZD020612 <= #1151
	out 3 "ФС02.01.06 промыт" <= #1149.regenerated
	out 4 "не удалось промыть" <= #1149.failToRegen
	#1153 ZD0212:SimpleValve(inputOpen: #1148, inputClose: NOT #1148, statusOpen: pin 8, statusClose: pin 9, reset: pin 4, timeToOpenClose: pin 10)
	out 9 "открыть ЗДЭ02.12" <= #1153.outputOpen
	out 10 "закрыть ЗДЭ02.12" <= #1153.outputClose
	out 11 "авария открытия ЗДЭ02.12" <= #1153.errorToOpen
	out 12 "авария закрытия ЗДЭ02.12" <= #1153.errorToClose
END_MACRO
#1154 DD2_DO.9 <= #1146.out 2
#1155 regeneratedFS020106 <= #1146.out 3
#1156 filterFailToRegen020106 <= #1146.out 4
#1157 DD2_DO.26 <= #1146.out 5
#1158 DD2_DO.27 <= #1146.out 6
#1159 errorToOpenZD0206 <= #1146.out 7
#1160 errorToCloseZD0206 <= #1146.out 8
#1161 DD3_DO.6 <= #1146.out 9
#1162 DD3_DO.7 <= #1146.out 10
#1163 errorToOpenZD0212 <= #1146.out 11
#1164 errorToCloseZD0212 <= #1146.out 12
